C03644=1019.173,313.342,359.557,170.379,50.215,159.769
C03645=1019.180,313.589,359.524,170.385,50.211,159.769
C03646=1019.186,313.837,359.491,170.391,50.208,159.770
C03647=1019.193,314.084,359.457,170.397,50.204,159.770
C03648=1019.200,314.331,359.424,170.404,50.201,159.770
C03649=1019.206,314.579,359.390,170.409,50.197,159.770
C03650=1019.212,314.826,359.357,170.415,50.194,159.770
C03651=1019.219,315.075,359.323,170.421,50.191,159.771
C03652=1019.226,315.322,359.290,170.427,50.187,159.771
C03653=1019.232,315.570,359.256,170.433,50.185,159.771
C03654=1019.239,315.817,359.223,170.439,50.181,159.771
C03655=1019.246,316.065,359.189,170.444,50.178,159.772
C03656=1019.252,316.312,359.156,170.451,50.175,159.772
C03657=1019.259,316.560,359.122,170.457,50.171,159.772
C03658=1019.265,316.807,359.088,170.463,50.168,159.772
C03659=1019.272,317.056,359.055,170.469,50.165,159.773
C03660=1019.279,317.303,359.021,170.475,50.162,159.773
C03661=1019.285,317.551,358.987,170.481,50.158,159.773
C03662=1019.292,317.798,358.954,170.487,50.156,159.773
C03663=1019.299,318.046,358.921,170.493,50.152,159.774
C03664=1019.306,318.294,358.887,170.500,50.149,159.774
C03665=1019.312,318.542,358.853,170.505,50.146,159.774
C03666=1019.319,318.789,358.819,170.512,50.143,159.775
C03667=1019.326,319.036,358.785,170.518,50.139,159.775
C03668=1019.333,319.284,358.752,170.523,50.136,159.775
C03669=1019.339,319.531,358.717,170.530,50.133,159.775
C03670=1019.346,319.779,358.684,170.535,50.130,159.776
C03671=1019.353,320.027,358.651,170.542,50.127,159.776
C03672=1019.360,320.274,358.617,170.549,50.124,159.776
C03673=1019.366,320.522,358.583,170.554,50.121,159.776
C03674=1019.374,320.770,358.549,170.561,50.118,159.777
C03675=1019.381,321.017,358.515,170.566,50.115,159.777
C03676=1019.387,321.264,358.482,170.572,50.111,159.777
C03677=1019.394,321.512,358.447,170.579,50.108,159.778
C03678=1019.401,321.760,358.413,170.585,50.106,159.778
C03679=1019.408,322.009,358.379,170.591,50.103,159.778
C03680=1019.415,322.258,358.344,170.598,50.099,159.779
C03681=1019.422,322.507,358.311,170.603,50.096,159.779
C03682=1019.429,322.756,358.276,170.610,50.093,159.779
C03683=1019.437,323.004,358.242,170.617,50.090,159.780
C03684=1019.443,323.252,358.208,170.622,50.088,159.780
C03685=1019.450,323.498,358.174,170.629,50.084,159.780
C03686=1019.457,323.746,358.141,170.635,50.081,159.781
C03687=1019.463,323.994,358.106,170.642,50.078,159.781
C03688=1019.471,324.241,358.072,170.647,50.075,159.781
C03689=1019.478,324.489,358.038,170.654,50.072,159.782
C03690=1019.485,324.737,358.004,170.661,50.069,159.782
C03691=1019.492,324.985,357.970,170.666,50.066,159.782
C03692=1019.499,325.232,357.935,170.673,50.063,159.783
C03693=1019.506,325.479,357.901,170.680,50.060,159.783
C03694=1019.514,325.727,357.867,170.685,50.058,159.783
C03695=1019.520,325.974,357.832,170.692,50.055,159.784
C03696=1019.528,326.222,357.798,170.699,50.052,159.784
C03697=1019.535,326.469,357.764,170.704,50.049,159.784
C03698=1019.542,326.717,357.730,170.711,50.046,159.785
C03699=1019.548,326.964,357.694,170.718,50.043,159.785
C03700=1019.555,327.212,357.661,170.724,50.041,159.786
C03701=1019.562,327.459,357.625,170.730,50.038,159.786
C03702=1019.569,327.707,357.590,170.737,50.035,159.787
C03703=1019.576,327.954,357.556,170.743,50.032,159.787
C03704=1019.583,328.202,357.521,170.750,50.030,159.787
C03705=1019.590,328.449,357.486,170.756,50.027,159.788
C03706=1019.597,328.697,357.451,170.762,50.024,159.788
C03707=1019.604,328.944,357.417,170.769,50.022,159.789
C03708=1019.610,329.192,357.382,170.776,50.019,159.789
C03709=1019.617,329.439,357.347,170.781,50.016,159.789
C03710=1019.625,329.686,357.312,170.788,50.014,159.790
C03711=1019.632,329.933,357.277,170.795,50.011,159.790
C03712=1019.639,330.182,357.242,170.801,50.009,159.791
C03713=1019.645,330.429,357.207,170.808,50.006,159.791
C03714=1019.653,330.676,357.173,170.814,50.003,159.792
C03715=1019.660,330.924,357.138,170.821,50.000,159.792
C03716=1019.666,331.171,357.103,170.827,49.998,159.793
C03717=1019.673,331.419,357.067,170.834,49.995,159.793
C03718=1019.681,331.666,357.033,170.841,49.992,159.793
C03719=1019.688,331.914,356.997,170.847,49.990,159.794
C03720=1019.695,332.161,356.962,170.853,49.987,159.794
C03721=1019.702,332.408,356.928,170.860,49.985,159.795
C03722=1019.710,332.656,356.892,170.867,49.983,159.796
C03723=1019.716,332.904,356.857,170.873,49.980,159.796
C03724=1019.723,333.151,356.822,170.880,49.978,159.796
C03725=1019.730,333.398,356.786,170.887,49.975,159.797
C03726=1019.738,333.646,356.751,170.893,49.972,159.797
C03727=1019.744,333.893,356.715,170.900,49.970,159.798
C03728=1019.751,334.140,356.680,170.907,49.968,159.798
C03729=1019.758,334.387,356.644,170.914,49.965,159.799
C03730=1019.766,334.635,356.609,170.919,49.963,159.799
C03731=1019.772,334.883,356.574,170.926,49.960,159.800
C03732=1019.779,335.129,356.538,170.933,49.958,159.801
C03733=1019.787,335.377,356.502,170.939,49.956,159.801
C03734=1019.794,335.625,356.467,170.946,49.954,159.802
C03735=1019.801,335.872,356.431,170.953,49.951,159.802
C03736=1019.808,336.120,356.396,170.960,49.948,159.803
C03737=1019.815,336.366,356.360,170.966,49.946,159.803
C03738=1019.823,336.614,356.325,170.973,49.944,159.804
C03739=1019.830,336.860,356.290,170.980,49.941,159.804
C03740=1019.837,337.106,356.253,170.987,49.939,159.805
C03741=1019.844,337.352,356.218,170.993,49.937,159.805
C03742=1019.851,337.599,356.182,171.000,49.935,159.806
C03743=1019.859,337.844,356.148,171.007,49.932,159.806
C03744=1019.866,338.091,356.112,171.014,49.930,159.807
C03745=1019.873,338.336,356.076,171.020,49.928,159.808
C03746=1019.880,338.583,356.040,171.027,49.926,159.808
C03747=1019.887,338.830,356.004,171.034,49.923,159.809
C03748=1019.895,339.078,355.969,171.042,49.921,159.810
C03749=1019.902,339.324,355.933,171.049,49.919,159.810
C03750=1019.909,339.572,355.897,171.055,49.917,159.811
C03751=1019.917,339.819,355.861,171.062,49.915,159.811
C03752=1019.924,340.066,355.824,171.069,49.912,159.812
C03753=1019.931,340.315,355.789,171.076,49.911,159.813
C03754=1019.938,340.561,355.753,171.083,49.908,159.813
C03755=1019.946,340.809,355.717,171.089,49.906,159.814
C03756=1019.952,341.056,355.680,171.096,49.904,159.814
C03757=1019.960,341.303,355.644,171.104,49.902,159.815
C03758=1019.967,341.551,355.608,171.111,49.900,159.816
C03759=1019.974,341.797,355.572,171.118,49.897,159.816
C03760=1019.981,342.045,355.535,171.124,49.896,159.817
C03761=1019.989,342.293,355.499,171.131,49.894,159.817
C03762=1019.996,342.539,355.463,171.139,49.892,159.818
C03763=1020.004,342.786,355.426,171.146,49.889,159.819
C03764=1020.011,343.034,355.389,171.153,49.888,159.820
C03765=1020.018,343.281,355.353,171.160,49.885,159.820
C03766=1020.026,343.528,355.317,171.166,49.884,159.821
C03767=1020.033,343.776,355.280,171.173,49.882,159.821
C03768=1020.040,344.023,355.244,171.181,49.880,159.822
C03769=1020.048,344.269,355.208,171.188,49.877,159.823
C03770=1020.055,344.517,355.171,171.195,49.876,159.824
C03771=1020.062,344.765,355.135,171.202,49.873,159.824
C03772=1020.070,345.011,355.098,171.210,49.872,159.825
C03773=1020.077,345.259,355.061,171.217,49.870,159.826
C03774=1020.085,345.507,355.025,171.223,49.868,159.826
C03775=1020.092,345.753,354.988,171.230,49.866,159.827
C03776=1020.099,346.001,354.951,171.238,49.864,159.828
C03777=1020.107,346.247,354.914,171.245,49.862,159.828
C03778=1020.115,346.495,354.878,171.252,49.860,159.829
C03779=1020.122,346.742,354.841,171.260,49.859,159.830
C03780=1020.130,346.989,354.804,171.267,49.857,159.831
C03781=1020.138,347.236,354.767,171.274,49.854,159.831
C03782=1020.145,347.484,354.731,171.281,49.853,159.832
C03783=1020.152,347.731,354.693,171.289,49.851,159.833
C03784=1020.160,347.978,354.656,171.296,49.849,159.834
C03785=1020.167,348.226,354.619,171.304,49.848,159.834
C03786=1020.175,348.473,354.582,171.310,49.846,159.835
C03787=1020.182,348.720,354.545,171.317,49.844,159.836
C03788=1020.190,348.966,354.508,171.325,49.843,159.837
C03789=1020.197,349.214,354.471,171.332,49.841,159.837
C03790=1020.205,349.461,354.434,171.340,49.839,159.838
C03791=1020.212,349.708,354.397,171.347,49.837,159.839
C03792=1020.220,349.955,354.359,171.354,49.836,159.840
C03793=1020.228,350.202,354.322,171.362,49.834,159.841
C03794=1020.235,350.449,354.285,171.369,49.832,159.841
C03795=1020.242,350.696,354.247,171.376,49.830,159.842
C03796=1020.250,350.943,354.210,171.384,49.829,159.843
C03797=1020.257,351.190,354.173,171.392,49.828,159.844
C03798=1020.265,351.437,354.136,171.399,49.826,159.845
C03799=1020.272,351.682,354.099,171.406,49.824,159.845
C03800=1020.280,351.927,354.062,171.414,49.822,159.846
C03801=1020.288,352.171,354.025,171.421,49.821,159.847
C03802=1020.295,352.416,353.988,171.429,49.820,159.848
C03803=1020.302,352.661,353.951,171.436,49.818,159.849
C03804=1020.310,352.905,353.914,171.444,49.816,159.850
C03805=1020.318,353.150,353.876,171.451,49.814,159.850
C03806=1020.326,353.394,353.839,171.459,49.813,159.851
C03807=1020.334,353.641,353.802,171.466,49.811,159.852
C03808=1020.341,353.888,353.764,171.474,49.810,159.853
C03809=1020.350,354.135,353.726,171.481,49.809,159.854
C03810=1020.357,354.382,353.689,171.489,49.807,159.855
C03811=1020.364,354.629,353.651,171.497,49.806,159.856
C03812=1020.372,354.876,353.613,171.504,49.804,159.856
C03813=1020.380,355.124,353.575,171.512,49.803,159.857
C03814=1020.388,355.370,353.537,171.519,49.801,159.858
C03815=1020.395,355.617,353.500,171.527,49.800,159.859
C03816=1020.403,355.864,353.461,171.535,49.799,159.860
C03817=1020.410,356.111,353.424,171.542,49.797,159.861
C03818=1020.418,356.358,353.386,171.550,49.796,159.862
C03819=1020.427,356.605,353.348,171.557,49.794,159.863
C03820=1020.434,356.852,353.310,171.566,49.793,159.864
C03821=1020.442,357.099,353.271,171.574,49.792,159.865
C03822=1020.450,357.346,353.234,171.582,49.791,159.866
C03823=1020.458,357.594,353.195,171.589,49.789,159.866
C03824=1020.465,357.840,353.157,171.597,49.788,159.867
C03825=1020.474,358.087,353.119,171.604,49.787,159.868
C03826=1020.481,358.334,353.081,171.612,49.785,159.869
C03827=1020.490,358.581,353.043,171.620,49.784,159.870
C03828=1020.497,358.828,353.005,171.628,49.782,159.871
C03829=1020.505,359.075,352.966,171.636,49.781,159.872
C03830=1020.513,359.322,352.928,171.644,49.780,159.873
C03831=1020.521,359.569,352.889,171.652,49.779,159.874
C03832=1020.529,359.815,352.851,171.659,49.778,159.875
C03833=1020.537,360.063,352.812,171.667,49.777,159.876
C03834=1020.544,360.309,352.774,171.676,49.775,159.877
C03835=1020.552,360.556,352.735,171.684,49.774,159.878
C03836=1020.561,360.803,352.697,171.691,49.773,159.879
C03837=1020.568,361.050,352.659,171.699,49.772,159.880
C03838=1020.575,361.298,352.619,171.707,49.771,159.881
C03839=1020.583,361.543,352.580,171.716,49.770,159.882
C03840=1020.591,361.791,352.542,171.724,49.769,159.883
C03841=1020.600,362.038,352.503,171.732,49.768,159.884
C03842=1020.607,362.284,352.465,171.739,49.766,159.885
C03843=1020.616,362.531,352.426,171.747,49.765,159.886
C03844=1020.624,362.778,352.387,171.756,49.764,159.888
C03845=1020.631,363.025,352.349,171.764,49.763,159.889
C03846=1020.639,363.272,352.309,171.772,49.762,159.890
C03847=1020.647,363.519,352.270,171.780,49.762,159.891
C03848=1020.656,363.765,352.231,171.789,49.760,159.892
C03849=1020.664,364.013,352.192,171.796,49.759,159.893
C03850=1020.672,364.258,352.153,171.805,49.759,159.894
C03851=1020.680,364.506,352.115,171.813,49.757,159.895
C03852=1020.688,364.752,352.075,171.821,49.757,159.896
C03853=1020.696,365.000,352.036,171.829,49.755,159.897
C03854=1020.704,365.246,351.997,171.837,49.754,159.898
C03855=1020.713,365.493,351.958,171.846,49.753,159.899
C03856=1020.721,365.740,351.919,171.854,49.752,159.900
C03857=1020.729,365.986,351.880,171.862,49.752,159.902
C03858=1020.737,366.233,351.841,171.871,49.751,159.903
C03859=1020.745,366.482,351.801,171.879,49.750,159.904
C03860=1020.753,366.732,351.762,171.888,49.749,159.905
C03861=1020.762,366.981,351.722,171.896,49.748,159.906
C03862=1020.770,367.231,351.682,171.905,49.747,159.907
C03863=1020.779,367.478,351.643,171.913,49.746,159.908
C03864=1020.787,367.725,351.603,171.921,49.746,159.910
C03865=1020.796,367.971,351.564,171.930,49.744,159.911
C03866=1020.804,368.218,351.524,171.938,49.744,159.912
C03867=1020.812,368.465,351.485,171.947,49.743,159.913
C03868=1020.820,368.712,351.445,171.955,49.742,159.914
C03869=1020.828,368.958,351.406,171.963,49.742,159.916
C03870=1020.836,369.205,351.366,171.973,49.741,159.917
C03871=1020.845,369.451,351.326,171.981,49.741,159.918
C03872=1020.852,369.698,351.286,171.990,49.740,159.919
C03873=1020.861,369.945,351.246,171.998,49.739,159.920
C03874=1020.869,370.192,351.207,172.007,49.738,159.922
C03875=1020.877,370.437,351.167,172.015,49.738,159.923
C03876=1020.885,370.684,351.127,172.023,49.737,159.924
C03877=1020.894,370.932,351.087,172.033,49.736,159.925
C03878=1020.902,371.178,351.046,172.041,49.736,159.927
C03879=1020.911,371.425,351.007,172.050,49.735,159.928
C03880=1020.919,371.671,350.966,172.058,49.734,159.929
C03881=1020.927,371.917,350.927,172.067,49.734,159.930
C03882=1020.936,372.165,350.887,172.076,49.734,159.932
C03883=1020.944,372.411,350.847,172.085,49.733,159.933
C03884=1020.953,372.657,350.807,172.093,49.732,159.934
C03885=1020.961,372.905,350.766,172.102,49.732,159.936
C03886=1020.970,373.151,350.726,172.111,49.731,159.937
C03887=1020.978,373.397,350.686,172.120,49.731,159.938
C03888=1020.987,373.644,350.646,172.129,49.730,159.939
C03889=1020.995,373.890,350.605,172.137,49.730,159.941
C03890=1021.004,374.137,350.566,172.146,49.729,159.942
C03891=1021.012,374.384,350.525,172.155,49.729,159.943
C03892=1021.021,374.630,350.485,172.164,49.728,159.945
C03893=1021.030,374.877,350.444,172.173,49.728,159.946
C03894=1021.038,375.123,350.404,172.182,49.727,159.947
C03895=1021.047,375.371,350.364,172.191,49.727,159.949
C03896=1021.055,375.617,350.324,172.200,49.726,159.950
C03897=1021.064,375.864,350.283,172.209,49.726,159.951
C03898=1021.073,376.110,350.243,172.218,49.725,159.953
C03899=1021.081,376.357,350.202,172.227,49.725,159.954
C03900=1021.089,376.603,350.161,172.236,49.725,159.955
C03901=1021.098,376.850,350.120,172.245,49.725,159.957
C03902=1021.107,377.095,350.079,172.254,49.724,159.958
C03903=1021.116,377.342,350.038,172.263,49.724,159.960
C03904=1021.124,377.588,349.998,172.272,49.724,159.961
C03905=1021.132,377.835,349.957,172.282,49.723,159.962
C03906=1021.141,378.081,349.915,172.290,49.723,159.964
C03907=1021.150,378.328,349.875,172.300,49.723,159.965
C03908=1021.159,378.575,349.834,172.309,49.723,159.967
C03909=1021.167,378.820,349.792,172.319,49.723,159.968
C03910=1021.176,379.067,349.751,172.327,49.723,159.970
C03911=1021.185,379.314,349.710,172.337,49.722,159.971
C03912=1021.193,379.560,349.669,172.346,49.722,159.973
C03913=1021.202,379.806,349.628,172.356,49.722,159.974
C03914=1021.211,380.053,349.587,172.364,49.722,159.975
C03915=1021.219,380.299,349.546,172.374,49.722,159.977
C03916=1021.228,380.545,349.504,172.383,49.721,159.978
C03917=1021.237,380.792,349.463,172.393,49.721,159.980
C03918=1021.246,381.038,349.421,172.403,49.721,159.982
C03919=1021.256,381.310,349.376,172.412,49.721,159.983
C03920=1021.265,381.581,349.331,172.423,49.721,159.985
C03921=1021.276,381.852,349.285,172.434,49.721,159.986
C03922=1021.285,382.124,349.239,172.444,49.721,159.988
C03923=1021.294,382.370,349.197,172.453,49.721,159.990
C03924=1021.303,382.617,349.156,172.463,49.721,159.991
C03925=1021.313,382.863,349.115,172.473,49.721,159.993
C03926=1021.322,383.109,349.073,172.482,49.721,159.994
C03927=1021.331,383.356,349.031,172.492,49.720,159.996
C03928=1021.339,383.602,348.990,172.502,49.721,159.997
C03929=1021.348,383.848,348.948,172.511,49.720,159.999
C03930=1021.357,384.095,348.906,172.521,49.721,160.001
C03931=1021.367,384.341,348.865,172.531,49.721,160.002
C03932=1021.376,384.587,348.823,172.540,49.721,160.004
C03933=1021.385,384.833,348.782,172.550,49.721,160.005
C03934=1021.394,385.080,348.740,172.560,49.721,160.007
C03935=1021.403,385.326,348.698,172.570,49.721,160.008
C03936=1021.412,385.573,348.656,172.580,49.721,160.010
C03937=1021.421,385.819,348.614,172.589,49.721,160.012
C03938=1021.430,386.065,348.572,172.599,49.721,160.013
C03939=1021.440,386.311,348.529,172.609,49.721,160.015
C03940=1021.449,386.558,348.488,172.619,49.722,160.017
C03941=1021.458,386.803,348.445,172.629,49.722,160.018
C03942=1021.467,387.050,348.403,172.638,49.722,160.020
C03943=1021.477,387.296,348.361,172.648,49.723,160.022
C03944=1021.486,387.542,348.319,172.658,49.723,160.023
C03945=1021.495,387.788,348.277,172.669,49.723,160.025
C03946=1021.505,388.035,348.234,172.679,49.723,160.027
C03947=1021.513,388.281,348.192,172.689,49.723,160.028
C03948=1021.522,388.527,348.149,172.699,49.724,160.030
C03949=1021.531,388.773,348.107,172.709,49.724,160.032
C03950=1021.541,389.019,348.064,172.719,49.725,160.034
C03951=1021.550,389.265,348.021,172.729,49.725,160.035
C03952=1021.559,389.512,347.978,172.740,49.725,160.037
C03953=1021.569,389.757,347.936,172.749,49.725,160.039
C03954=1021.578,390.003,347.893,172.760,49.726,160.041
C03955=1021.588,390.250,347.850,172.770,49.726,160.042
C03956=1021.596,390.496,347.807,172.781,49.727,160.044
C03957=1021.606,390.742,347.765,172.791,49.727,160.046
C03958=1021.615,390.988,347.722,172.801,49.727,160.048
C03959=1021.625,391.234,347.679,172.811,49.728,160.050
C03960=1021.634,391.480,347.637,172.822,49.728,160.051
C03961=1021.644,391.727,347.593,172.832,49.729,160.053
C03962=1021.653,391.972,347.550,172.842,49.730,160.055
C03963=1021.663,392.218,347.508,172.853,49.730,160.057
C03964=1021.671,392.464,347.464,172.863,49.731,160.059
C03965=1021.682,392.710,347.421,172.873,49.731,160.060
C03966=1021.691,392.957,347.378,172.884,49.732,160.062
C03967=1021.700,393.202,347.334,172.895,49.732,160.064
C03968=1021.710,393.449,347.292,172.905,49.733,160.066
C03969=1021.720,393.694,347.248,172.916,49.734,160.068
C03970=1021.729,393.940,347.205,172.926,49.734,160.070
C03971=1021.739,394.186,347.162,172.937,49.734,160.072
C03972=1021.748,394.432,347.117,172.948,49.735,160.074
C03973=1021.758,394.679,347.075,172.958,49.736,160.076
C03974=1021.767,394.924,347.031,172.969,49.737,160.078
C03975=1021.777,395.170,346.987,172.979,49.737,160.079
C03976=1021.787,395.416,346.944,172.990,49.738,160.081
C03977=1021.796,395.663,346.901,173.001,49.739,160.083
C03978=1021.806,395.909,346.857,173.012,49.739,160.085
C03979=1021.819,396.217,346.802,173.026,49.740,160.088
C03980=1021.831,396.525,346.747,173.039,49.742,160.090
C03981=1021.843,396.834,346.693,173.053,49.743,160.093
C03982=1021.855,397.142,346.637,173.067,49.744,160.095
C03983=1021.865,397.388,346.593,173.078,49.744,160.097
C03984=1021.875,397.634,346.550,173.088,49.745,160.099
C03985=1021.884,397.880,346.506,173.100,49.746,160.101
C03986=1021.895,398.126,346.461,173.110,49.747,160.103
C03987=1021.904,398.372,346.417,173.122,49.748,160.105
C03988=1021.914,398.618,346.373,173.133,49.748,160.107
C03989=1021.924,398.863,346.329,173.144,49.750,160.110
C03990=1021.934,399.109,346.285,173.155,49.750,160.111
C03991=1021.944,399.355,346.241,173.167,49.751,160.114
C03992=1021.954,399.601,346.196,173.177,49.752,160.116
C03993=1021.964,399.847,346.151,173.189,49.753,160.118
C03994=1021.974,400.093,346.108,173.200,49.754,160.120
C03995=1021.984,400.338,346.063,173.212,49.755,160.122
C03996=1021.993,400.584,346.019,173.222,49.756,160.124
C03997=1022.004,400.830,345.974,173.234,49.757,160.126
C03998=1022.014,401.076,345.929,173.245,49.758,160.128
C03999=1022.024,401.321,345.885,173.257,49.759,160.131
C04000=1022.033,401.567,345.840,173.269,49.760,160.133
C04001=1022.043,401.814,345.795,173.279,49.762,160.135
C04002=1022.053,402.059,345.751,173.291,49.763,160.137
C04003=1022.063,402.304,345.706,173.302,49.764,160.139
C04004=1022.074,402.550,345.661,173.314,49.765,160.141
C04005=1022.084,402.795,345.616,173.326,49.766,160.144
C04006=1022.093,403.041,345.571,173.338,49.767,160.146
C04007=1022.104,403.287,345.526,173.349,49.768,160.148
C04008=1022.114,403.532,345.481,173.361,49.769,160.150
C04009=1022.125,403.778,345.436,173.373,49.770,160.152
C04010=1022.134,404.024,345.391,173.385,49.772,160.155
C04011=1022.145,404.270,345.345,173.396,49.773,160.157
C04012=1022.155,404.515,345.301,173.408,49.774,160.159
C04013=1022.165,404.761,345.255,173.420,49.776,160.162
C04014=1022.176,405.006,345.210,173.431,49.777,160.164
C04015=1022.186,405.252,345.165,173.443,49.778,160.166
C04016=1022.196,405.497,345.120,173.455,49.779,160.168
C04017=1022.206,405.743,345.075,173.467,49.781,160.171
C04018=1022.217,405.989,345.029,173.479,49.782,160.173
C04019=1022.227,406.235,344.983,173.491,49.783,160.175
C04020=1022.237,406.480,344.938,173.503,49.785,160.178
C04021=1022.249,406.725,344.893,173.516,49.786,160.180
C04022=1022.259,406.971,344.847,173.527,49.787,160.182
C04023=1022.270,407.217,344.801,173.539,49.789,160.185
C04024=1022.280,407.462,344.756,173.551,49.790,160.187
C04025=1022.290,407.708,344.710,173.563,49.792,160.190
C04026=1022.301,407.954,344.665,173.576,49.793,160.192
C04027=1022.312,408.199,344.620,173.588,49.795,160.194
C04028=1022.323,408.445,344.574,173.600,49.796,160.197
C04029=1022.333,408.690,344.528,173.613,49.798,160.199
C04030=1022.344,408.936,344.482,173.625,49.799,160.202
C04031=1022.354,409.181,344.436,173.637,49.801,160.204
C04032=1022.365,409.427,344.390,173.650,49.802,160.207
C04033=1022.376,409.672,344.343,173.662,49.803,160.209
C04034=1022.387,409.918,344.297,173.675,49.806,160.212
C04035=1022.397,410.163,344.252,173.688,49.807,160.214
C04036=1022.407,410.408,344.204,173.700,49.808,160.216
C04037=1022.418,410.654,344.158,173.712,49.811,160.219
C04038=1022.429,410.899,344.112,173.725,49.812,160.222
C04039=1022.444,411.231,344.049,173.743,49.814,160.225
C04040=1022.458,411.561,343.987,173.760,49.816,160.228
C04041=1022.473,411.893,343.924,173.776,49.819,160.232
C04042=1022.488,412.224,343.861,173.794,49.821,160.235
C04043=1022.498,412.470,343.814,173.807,49.823,160.238
C04044=1022.509,412.715,343.768,173.819,49.825,160.241
C04045=1022.520,412.960,343.721,173.833,49.826,160.243
C04046=1022.531,413.206,343.674,173.846,49.828,160.246
C04047=1022.542,413.451,343.628,173.858,49.830,160.248
C04048=1022.554,413.697,343.581,173.871,49.831,160.251
C04049=1022.564,413.942,343.533,173.885,49.833,160.254
C04050=1022.575,414.187,343.487,173.897,49.835,160.256
C04051=1022.587,414.433,343.440,173.911,49.837,160.259
C04052=1022.598,414.678,343.393,173.924,49.839,160.262
C04053=1022.609,414.923,343.346,173.937,49.840,160.264
C04054=1022.621,415.169,343.299,173.950,49.842,160.267
C04055=1022.631,415.414,343.252,173.964,49.845,160.270
C04056=1022.643,415.659,343.204,173.977,49.847,160.273
C04057=1022.653,415.905,343.157,173.990,49.848,160.275
C04058=1022.665,416.150,343.109,174.004,49.851,160.278
C04059=1022.676,416.395,343.062,174.017,49.852,160.281
C04060=1022.687,416.640,343.014,174.031,49.855,160.284
C04061=1022.698,416.886,342.967,174.044,49.857,160.286
C04062=1022.709,417.131,342.919,174.057,49.859,160.289
C04063=1022.721,417.375,342.872,174.071,49.861,160.292
C04064=1022.731,417.621,342.824,174.085,49.863,160.295
C04065=1022.743,417.866,342.776,174.098,49.865,160.298
C04066=1022.755,418.111,342.729,174.112,49.867,160.301
C04067=1022.766,418.357,342.680,174.126,49.869,160.304
C04068=1022.778,418.602,342.633,174.140,49.871,160.306
C04069=1022.788,418.847,342.585,174.154,49.873,160.309
C04070=1022.800,419.092,342.537,174.168,49.875,160.312
C04071=1022.811,419.337,342.489,174.182,49.878,160.315
C04072=1022.823,419.582,342.441,174.195,49.880,160.318
C04073=1022.835,419.827,342.393,174.209,49.882,160.321
C04074=1022.846,420.072,342.345,174.224,49.884,160.324
C04075=1022.858,420.317,342.297,174.238,49.886,160.327
C04076=1022.870,420.563,342.248,174.251,49.888,160.330
C04077=1022.882,420.808,342.200,174.265,49.891,160.333
C04078=1022.894,421.053,342.153,174.280,49.893,160.336
C04079=1022.905,421.298,342.104,174.294,49.895,160.339
C04080=1022.917,421.543,342.056,174.308,49.898,160.342
C04081=1022.929,421.789,342.007,174.323,49.900,160.345
C04082=1022.940,422.034,341.958,174.337,49.902,160.348
C04083=1022.952,422.278,341.910,174.352,49.905,160.351
C04084=1022.964,422.523,341.861,174.366,49.907,160.354
C04085=1022.975,422.769,341.812,174.380,49.910,160.357
C04086=1022.987,423.013,341.764,174.395,49.912,160.360
C04087=1022.999,423.258,341.715,174.409,49.915,160.364
C04088=1023.011,423.503,341.665,174.424,49.917,160.367
C04089=1023.023,423.748,341.617,174.439,49.919,160.370
C04090=1023.034,423.993,341.568,174.453,49.922,160.373
C04091=1023.047,424.238,341.519,174.469,49.924,160.376
C04092=1023.059,424.483,341.470,174.483,49.927,160.379
C04093=1023.071,424.728,341.421,174.498,49.929,160.382
C04094=1023.083,424.972,341.372,174.513,49.932,160.386
C04095=1023.095,425.217,341.322,174.528,49.935,160.389
C04096=1023.107,425.463,341.273,174.543,49.937,160.392
C04097=1023.120,425.708,341.224,174.558,49.940,160.395
C04098=1023.131,425.952,341.174,174.573,49.942,160.399
C04099=1023.145,426.222,341.120,174.590,49.945,160.402
C04100=1023.158,426.491,341.065,174.607,49.948,160.406
C04101=1023.171,426.761,341.010,174.623,49.951,160.410
C04102=1023.185,427.031,340.956,174.640,49.954,160.413
C04103=1023.197,427.275,340.906,174.655,49.957,160.417
C04104=1023.209,427.520,340.856,174.670,49.960,160.420
C04105=1023.221,427.764,340.806,174.686,49.963,160.423
C04106=1023.234,428.009,340.756,174.701,49.965,160.427
C04107=1023.246,428.254,340.706,174.717,49.968,160.430
C04108=1023.258,428.499,340.656,174.732,49.971,160.434
C04109=1023.271,428.744,340.605,174.749,49.974,160.437
C04110=1023.284,428.988,340.556,174.764,49.977,160.441
C04111=1023.296,429.233,340.506,174.780,49.979,160.444
C04112=1023.308,429.478,340.456,174.796,49.982,160.447
C04113=1023.321,429.722,340.405,174.811,49.985,160.451
C04114=1023.333,429.967,340.355,174.827,49.988,160.454
C04115=1023.346,430.212,340.305,174.843,49.990,160.458
C04116=1023.358,430.456,340.254,174.859,49.994,160.461
C04117=1023.371,430.700,340.204,174.875,49.997,160.465
C04118=1023.384,430.945,340.154,174.892,50.000,160.469
C04119=1023.397,431.190,340.103,174.907,50.003,160.472
C04120=1023.409,431.434,340.052,174.924,50.006,160.476
C04121=1023.422,431.678,340.002,174.940,50.008,160.479
C04122=1023.434,431.923,339.951,174.956,50.012,160.483
C04123=1023.448,432.168,339.901,174.973,50.015,160.487
C04124=1023.461,432.413,339.850,174.989,50.017,160.490
C04125=1023.474,432.657,339.799,175.005,50.021,160.494
C04126=1023.487,432.901,339.748,175.022,50.024,160.497
C04127=1023.500,433.146,339.697,175.038,50.027,160.501
C04128=1023.513,433.390,339.646,175.055,50.030,160.505
C04129=1023.525,433.636,339.594,175.072,50.033,160.509
C04130=1023.538,433.879,339.543,175.088,50.036,160.512
C04131=1023.551,434.124,339.492,175.105,50.040,160.516
C04132=1023.564,434.369,339.440,175.122,50.043,160.520
C04133=1023.577,434.612,339.389,175.139,50.046,160.524
C04134=1023.591,434.857,339.338,175.156,50.049,160.528
C04135=1023.603,435.101,339.286,175.172,50.053,160.531
C04136=1023.617,435.345,339.234,175.190,50.056,160.535
C04137=1023.630,435.590,339.183,175.206,50.059,160.539
C04138=1023.644,435.834,339.131,175.224,50.062,160.543
C04139=1023.660,436.152,339.064,175.247,50.067,160.548
C04140=1023.678,436.468,338.997,175.269,50.071,160.553
C04141=1023.695,436.786,338.929,175.291,50.076,160.558
C04142=1023.713,437.103,338.862,175.314,50.080,160.563
C04143=1023.726,437.347,338.810,175.332,50.083,160.567
C04144=1023.740,437.592,338.758,175.349,50.087,160.571
C04145=1023.753,437.836,338.706,175.366,50.090,160.575
C04146=1023.766,438.080,338.653,175.384,50.093,160.579
C04147=1023.780,438.324,338.601,175.402,50.097,160.584
C04148=1023.794,438.568,338.548,175.420,50.101,160.587
C04149=1023.807,438.812,338.496,175.438,50.104,160.592
C04150=1023.820,439.056,338.443,175.456,50.108,160.596
C04151=1023.834,439.301,338.391,175.474,50.111,160.600
C04152=1023.848,439.545,338.338,175.492,50.115,160.604
C04153=1023.862,439.788,338.286,175.510,50.118,160.608
C04154=1023.875,440.032,338.232,175.528,50.122,160.612
C04155=1023.889,440.277,338.180,175.547,50.126,160.617
C04156=1023.903,440.521,338.128,175.565,50.130,160.621
C04157=1023.918,440.765,338.075,175.583,50.133,160.625
C04158=1023.931,441.009,338.022,175.602,50.137,160.629
C04159=1023.946,441.268,337.966,175.621,50.141,160.634
C04160=1023.961,441.529,337.909,175.641,50.144,160.638
C04161=1023.976,441.789,337.852,175.661,50.148,160.643
C04162=1023.991,442.047,337.795,175.680,50.152,160.647
C04163=1023.596,440.124,337.880,175.526,50.187,160.632
C04164=1023.583,439.880,337.933,175.508,50.184,160.628
C04165=1023.569,439.636,337.986,175.490,50.180,160.624
C04166=1023.555,439.391,338.038,175.472,50.177,160.620
C04167=1023.541,439.147,338.091,175.453,50.174,160.615
C04168=1023.528,438.903,338.144,175.436,50.170,160.611
C04169=1023.514,438.659,338.196,175.417,50.167,160.607
C04170=1023.501,438.415,338.248,175.400,50.163,160.603
C04171=1023.487,438.171,338.300,175.382,50.160,160.599
C04172=1023.474,437.927,338.353,175.364,50.157,160.595
C04173=1023.460,437.682,338.406,175.347,50.154,160.591
C04174=1023.446,437.438,338.458,175.329,50.150,160.587
C04175=1023.433,437.194,338.509,175.311,50.147,160.583
C04176=1023.419,436.949,338.561,175.294,50.144,160.579
C04177=1023.406,436.705,338.613,175.276,50.140,160.575
C04178=1023.393,436.461,338.665,175.259,50.137,160.571
C04179=1023.379,436.217,338.717,175.242,50.133,160.567
C04180=1023.366,435.973,338.769,175.225,50.130,160.564
C04181=1023.353,435.728,338.820,175.207,50.127,160.560
C04182=1023.340,435.483,338.872,175.190,50.124,160.556
C04183=1023.327,435.240,338.924,175.173,50.121,160.552
C04184=1023.314,434.995,338.975,175.156,50.118,160.548
C04185=1023.300,434.751,339.027,175.139,50.115,160.544
C04186=1023.287,434.506,339.078,175.122,50.111,160.540
C04187=1023.274,434.262,339.129,175.105,50.108,160.537
C04188=1023.261,434.017,339.181,175.088,50.105,160.533
C04189=1023.248,433.773,339.231,175.071,50.102,160.529
C04190=1023.235,433.529,339.283,175.055,50.099,160.525
C04191=1023.222,433.285,339.334,175.038,50.096,160.522
C04192=1023.209,433.040,339.385,175.021,50.093,160.518
C04193=1023.197,432.795,339.437,175.005,50.090,160.514
C04194=1023.184,432.551,339.488,174.988,50.087,160.511
C04195=1023.170,432.306,339.538,174.972,50.084,160.507
C04196=1023.158,432.062,339.589,174.956,50.081,160.503
C04197=1023.144,431.817,339.640,174.939,50.078,160.500
C04198=1023.132,431.572,339.690,174.923,50.075,160.496
C04199=1023.119,431.328,339.741,174.906,50.072,160.492
C04200=1023.106,431.083,339.792,174.891,50.069,160.489
C04201=1023.093,430.839,339.842,174.874,50.067,160.485
C04202=1023.081,430.595,339.893,174.858,50.064,160.482
C04203=1023.068,430.350,339.943,174.841,50.061,160.478
C04204=1023.054,430.093,339.995,174.825,50.058,160.475
C04205=1023.042,429.838,340.048,174.809,50.055,160.471
C04206=1023.028,429.583,340.101,174.792,50.052,160.467
C04207=1023.015,429.327,340.153,174.775,50.050,160.464
C04208=1023.003,429.082,340.203,174.760,50.047,160.460
C04209=1022.991,428.837,340.253,174.744,50.044,160.457
C04210=1022.978,428.592,340.303,174.728,50.041,160.453
C04211=1022.966,428.348,340.353,174.712,50.039,160.450
C04212=1022.954,428.103,340.404,174.697,50.036,160.447
C04213=1022.941,427.858,340.454,174.681,50.033,160.443
C04214=1022.928,427.613,340.503,174.666,50.031,160.440
C04215=1022.916,427.369,340.553,174.650,50.028,160.436
C04216=1022.900,427.040,340.620,174.630,50.025,160.432
C04217=1022.884,426.711,340.687,174.609,50.020,160.427
C04218=1022.867,426.383,340.753,174.589,50.017,160.423
C04219=1022.852,426.055,340.820,174.568,50.014,160.419
C04220=1022.839,425.810,340.869,174.554,50.011,160.416
C04221=1022.827,425.565,340.919,174.538,50.008,160.412
C04222=1022.816,425.320,340.968,174.523,50.006,160.409
C04223=1022.803,425.075,341.018,174.508,50.004,160.406
C04224=1022.791,424.830,341.066,174.493,50.001,160.402
C04225=1022.779,424.586,341.116,174.479,49.999,160.399
C04226=1022.767,424.340,341.165,174.463,49.996,160.396
C04227=1022.755,424.096,341.213,174.448,49.994,160.393
C04228=1022.743,423.850,341.263,174.434,49.992,160.390
C04229=1022.731,423.606,341.311,174.419,49.989,160.387
C04230=1022.719,423.361,341.360,174.404,49.987,160.383
C04231=1022.707,423.116,341.410,174.390,49.984,160.380
C04232=1022.695,422.871,341.458,174.375,49.982,160.377
C04233=1022.684,422.626,341.507,174.361,49.980,160.374
C04234=1022.672,422.380,341.556,174.346,49.978,160.371
C04235=1022.660,422.136,341.604,174.332,49.975,160.368
C04236=1022.649,421.891,341.653,174.317,49.973,160.365
C04237=1022.637,421.646,341.701,174.303,49.970,160.362
C04238=1022.625,421.401,341.750,174.288,49.969,160.359
C04239=1022.614,421.155,341.798,174.275,49.966,160.356
C04240=1022.602,420.911,341.847,174.260,49.965,160.353
C04241=1022.590,420.666,341.895,174.246,49.962,160.350
C04242=1022.579,420.421,341.943,174.232,49.960,160.347
C04243=1022.567,420.175,341.991,174.217,49.958,160.344
C04244=1022.555,419.931,342.040,174.203,49.955,160.341
C04245=1022.544,419.686,342.087,174.189,49.953,160.338
C04246=1022.532,419.441,342.135,174.176,49.951,160.335
C04247=1022.521,419.195,342.183,174.161,49.950,160.332
C04248=1022.509,418.950,342.231,174.147,49.947,160.329
C04249=1022.498,418.705,342.279,174.134,49.945,160.326
C04250=1022.486,418.460,342.327,174.120,49.943,160.324
C04251=1022.474,418.215,342.375,174.106,49.941,160.321
C04252=1022.463,417.969,342.422,174.093,49.939,160.318
C04253=1022.451,417.724,342.470,174.078,49.937,160.315
C04254=1022.441,417.479,342.518,174.064,49.935,160.312
C04255=1022.429,417.234,342.566,174.051,49.933,160.309
C04256=1022.418,416.988,342.613,174.037,49.932,160.307
C04257=1022.406,416.743,342.661,174.023,49.929,160.304
C04258=1022.395,416.498,342.707,174.010,49.928,160.301
C04259=1022.384,416.253,342.756,173.997,49.926,160.298
C04260=1022.373,416.007,342.803,173.984,49.923,160.295
C04261=1022.362,415.762,342.851,173.970,49.922,160.293
C04262=1022.351,415.517,342.898,173.957,49.920,160.290
C04263=1022.340,415.272,342.945,173.944,49.918,160.287
C04264=1022.329,415.026,342.993,173.930,49.916,160.285
C04265=1022.318,414.781,343.039,173.917,49.915,160.282
C04266=1022.306,414.536,343.086,173.903,49.913,160.279
C04267=1022.295,414.291,343.133,173.890,49.911,160.277
C04268=1022.284,414.045,343.180,173.878,49.909,160.274
C04269=1022.273,413.800,343.226,173.864,49.907,160.271
C04270=1022.262,413.554,343.274,173.851,49.906,160.268
C04271=1022.251,413.309,343.321,173.837,49.904,160.266
C04272=1022.240,413.063,343.368,173.825,49.902,160.263
C04273=1022.229,412.818,343.414,173.812,49.901,160.261
C04274=1022.218,412.573,343.460,173.799,49.899,160.258
C04275=1022.207,412.328,343.507,173.787,49.898,160.256
C04276=1022.192,411.994,343.571,173.769,49.895,160.252
C04277=1022.178,411.661,343.633,173.752,49.893,160.248
C04278=1022.163,411.326,343.697,173.734,49.891,160.245
C04279=1022.149,410.993,343.760,173.717,49.888,160.241
C04280=1022.138,410.748,343.806,173.704,49.887,160.239
C04281=1022.127,410.501,343.853,173.692,49.886,160.237
C04282=1022.116,410.256,343.899,173.678,49.884,160.234
C04283=1022.105,410.011,343.945,173.666,49.882,160.231
C04284=1022.094,409.766,343.992,173.653,49.881,160.229
C04285=1022.084,409.520,344.038,173.641,49.880,160.227
C04286=1022.074,409.274,344.084,173.628,49.878,160.224
C04287=1022.063,409.029,344.130,173.616,49.877,160.222
C04288=1022.053,408.783,344.176,173.604,49.875,160.219
C04289=1022.041,408.538,344.221,173.591,49.874,160.217
C04290=1022.031,408.292,344.267,173.579,49.873,160.214
C04291=1022.020,408.047,344.313,173.567,49.871,160.212
C04292=1022.010,407.802,344.359,173.554,49.870,160.210
C04293=1021.999,407.556,344.405,173.542,49.868,160.207
C04294=1021.989,407.310,344.450,173.531,49.867,160.205
C04295=1021.978,407.065,344.495,173.518,49.866,160.202
C04296=1021.967,406.819,344.541,173.506,49.864,160.200
C04297=1021.957,406.574,344.586,173.494,49.863,160.198
C04298=1021.947,406.328,344.632,173.482,49.862,160.195
C04299=1021.936,406.082,344.678,173.469,49.861,160.193
C04300=1021.926,405.836,344.723,173.457,49.860,160.191
C04301=1021.915,405.592,344.768,173.445,49.858,160.188
C04302=1021.905,405.345,344.813,173.434,49.857,160.186
C04303=1021.894,405.100,344.859,173.422,49.856,160.184
C04304=1021.884,404.854,344.904,173.410,49.854,160.182
C04305=1021.874,404.608,344.949,173.398,49.853,160.179
C04306=1021.863,404.363,344.994,173.386,49.853,160.177
C04307=1021.853,404.117,345.039,173.374,49.851,160.175
C04308=1021.843,403.872,345.084,173.362,49.850,160.173
C04309=1021.833,403.625,345.129,173.350,49.849,160.170
C04310=1021.823,403.381,345.175,173.339,49.848,160.168
C04311=1021.813,403.134,345.220,173.327,49.847,160.166
C04312=1021.802,402.889,345.264,173.315,49.846,160.164
C04313=1021.792,402.644,345.309,173.303,49.845,160.161
C04314=1021.782,402.397,345.354,173.292,49.844,160.159
C04315=1021.772,402.152,345.399,173.281,49.842,160.157
C04316=1021.763,401.906,345.444,173.270,49.842,160.155
C04317=1021.752,401.660,345.489,173.258,49.841,160.153
C04318=1021.742,401.415,345.533,173.247,49.840,160.151
C04319=1021.732,401.170,345.578,173.235,49.839,160.148
C04320=1021.723,400.923,345.622,173.223,49.838,160.146
C04321=1021.712,400.677,345.667,173.212,49.837,160.144
C04322=1021.702,400.432,345.711,173.200,49.836,160.142
C04323=1021.693,400.186,345.755,173.190,49.835,160.140
C04324=1021.683,399.940,345.800,173.178,49.834,160.138
C04325=1021.672,399.695,345.845,173.167,49.833,160.136
C04326=1021.663,399.449,345.889,173.155,49.832,160.134
C04327=1021.653,399.203,345.933,173.144,49.832,160.132
C04328=1021.643,398.957,345.977,173.133,49.830,160.130
C04329=1021.633,398.711,346.021,173.122,49.830,160.128
C04330=1021.623,398.466,346.066,173.111,49.829,160.125
C04331=1021.613,398.219,346.110,173.099,49.828,160.123
C04332=1021.604,397.973,346.154,173.089,49.827,160.121
C04333=1021.594,397.727,346.197,173.077,49.827,160.119
C04334=1021.584,397.482,346.242,173.066,49.826,160.117
C04335=1021.574,397.236,346.286,173.056,49.825,160.115
C04336=1021.562,396.925,346.341,173.042,49.824,160.113
C04337=1021.549,396.614,346.396,173.028,49.823,160.110
C04338=1021.537,396.303,346.452,173.014,49.822,160.108
C04339=1021.525,395.992,346.507,173.000,49.822,160.105
C04340=1021.514,395.746,346.551,172.990,49.821,160.104
C04341=1021.506,395.500,346.594,172.979,49.821,160.102
C04342=1021.496,395.255,346.637,172.967,49.820,160.100
C04343=1021.486,395.009,346.681,172.957,49.819,160.098
C04344=1021.476,394.763,346.725,172.946,49.819,160.096
C04345=1021.466,394.516,346.768,172.936,49.818,160.094
C04346=1021.458,394.271,346.811,172.924,49.818,160.092
C04347=1021.447,394.025,346.855,172.914,49.817,160.090
C04348=1021.438,393.778,346.898,172.903,49.817,160.088
C04349=1021.429,393.533,346.941,172.893,49.816,160.086
C04350=1021.419,393.287,346.984,172.882,49.816,160.084
C04351=1021.410,393.040,347.028,172.871,49.815,160.082
C04352=1021.400,392.795,347.071,172.862,49.814,160.081
C04353=1021.391,392.549,347.115,172.850,49.814,160.079
C04354=1021.382,392.303,347.157,172.840,49.814,160.077
C04355=1021.372,392.056,347.200,172.829,49.813,160.075
C04356=1021.362,391.811,347.244,172.819,49.813,160.073
C04357=1021.353,391.565,347.287,172.809,49.812,160.072
C04358=1021.343,391.318,347.329,172.798,49.812,160.070
C04359=1021.334,391.072,347.372,172.788,49.811,160.068
C04360=1021.324,390.826,347.415,172.778,49.811,160.066
C04361=1021.315,390.580,347.457,172.767,49.811,160.064
C04362=1021.306,390.333,347.500,172.757,49.810,160.063
C04363=1021.296,390.088,347.544,172.747,49.810,160.061
C04364=1021.287,389.842,347.585,172.736,49.810,160.059
C04365=1021.278,389.595,347.628,172.726,49.810,160.057
C04366=1021.269,389.349,347.671,172.716,49.810,160.056
C04367=1021.260,389.104,347.714,172.706,49.809,160.054
C04368=1021.250,388.857,347.756,172.695,49.809,160.052
C04369=1021.241,388.611,347.799,172.685,49.809,160.050
C04370=1021.231,388.366,347.841,172.675,49.808,160.049
C04371=1021.223,388.118,347.884,172.666,49.808,160.047
C04372=1021.213,387.873,347.926,172.656,49.808,160.045
C04373=1021.204,387.627,347.969,172.645,49.808,160.044
C04374=1021.195,387.380,348.011,172.635,49.808,160.042
C04375=1021.185,387.134,348.053,172.625,49.807,160.040
C04376=1021.177,386.888,348.095,172.616,49.808,160.039
C04377=1021.167,386.642,348.137,172.606,49.807,160.037
C04378=1021.158,386.396,348.179,172.596,49.807,160.035
C04379=1021.149,386.150,348.222,172.585,49.807,160.034
C04380=1021.140,385.903,348.264,172.575,49.807,160.032
C04381=1021.130,385.657,348.306,172.566,49.807,160.030
C04382=1021.121,385.411,348.348,172.556,49.807,160.029
C04383=1021.112,385.164,348.390,172.546,49.807,160.027
C04384=1021.104,384.918,348.431,172.536,49.807,160.026
C04385=1021.095,384.672,348.473,172.526,49.807,160.024
C04386=1021.086,384.425,348.515,172.517,49.807,160.022
C04387=1021.077,384.179,348.556,172.507,49.807,160.021
C04388=1021.067,383.933,348.598,172.497,49.807,160.019
C04389=1021.058,383.687,348.640,172.488,49.807,160.018
C04390=1021.049,383.441,348.682,172.478,49.807,160.016
C04391=1021.040,383.194,348.723,172.469,49.807,160.015
C04392=1021.031,382.947,348.764,172.459,49.807,160.013
C04393=1021.022,382.701,348.806,172.449,49.807,160.011
C04394=1021.013,382.455,348.847,172.440,49.808,160.010
C04395=1021.004,382.209,348.889,172.430,49.808,160.009
C04396=1020.994,381.934,348.935,172.419,49.808,160.007
C04397=1020.984,381.661,348.981,172.408,49.808,160.005
C04398=1020.975,381.387,349.027,172.398,49.809,160.003
C04399=1020.964,381.113,349.073,172.387,49.809,160.002
C04400=1020.956,380.867,349.114,172.379,49.809,160.000
C04401=1020.947,380.621,349.156,172.369,49.809,159.999
C04402=1020.938,380.374,349.196,172.360,49.809,159.997
C04403=1020.929,380.128,349.238,172.350,49.810,159.996
C04404=1020.920,379.882,349.279,172.341,49.810,159.994
C04405=1020.912,379.635,349.320,172.331,49.810,159.993
C04406=1020.903,379.389,349.362,172.321,49.811,159.991
C04407=1020.894,379.142,349.403,172.313,49.811,159.990
C04408=1020.885,378.896,349.443,172.303,49.811,159.989
C04409=1020.876,378.649,349.485,172.294,49.811,159.987
C04410=1020.868,378.403,349.525,172.284,49.812,159.986
C04411=1020.859,378.157,349.567,172.275,49.812,159.984
C04412=1020.851,377.910,349.608,172.266,49.812,159.983
C04413=1020.842,377.664,349.648,172.257,49.813,159.981
C04414=1020.833,377.417,349.689,172.248,49.813,159.980
C04415=1020.825,377.171,349.730,172.238,49.813,159.979
C04416=1020.816,376.924,349.771,172.230,49.813,159.977
C04417=1020.808,376.678,349.812,172.221,49.814,159.976
C04418=1020.800,376.431,349.853,172.211,49.814,159.974
C04419=1020.791,376.185,349.893,172.202,49.815,159.973
C04420=1020.782,375.938,349.934,172.193,49.815,159.972
C04421=1020.774,375.692,349.974,172.184,49.816,159.970
C04422=1020.765,375.445,350.015,172.175,49.816,159.969
C04423=1020.756,375.199,350.055,172.167,49.817,159.968
C04424=1020.748,374.952,350.096,172.157,49.817,159.966
C04425=1020.739,374.705,350.135,172.148,49.818,159.965
C04426=1020.731,374.458,350.176,172.139,49.818,159.964
C04427=1020.722,374.212,350.217,172.130,49.819,159.962
C04428=1020.714,373.966,350.257,172.121,49.820,159.961
C04429=1020.705,373.719,350.297,172.112,49.820,159.960
C04430=1020.697,373.473,350.337,172.104,49.821,159.958
C04431=1020.688,373.225,350.377,172.095,49.822,159.957
C04432=1020.680,372.979,350.418,172.086,49.822,159.956
C04433=1020.671,372.733,350.458,172.077,49.823,159.955
C04434=1020.663,372.486,350.498,172.068,49.823,159.953
C04435=1020.654,372.239,350.538,172.060,49.824,159.952
C04436=1020.646,371.993,350.578,172.050,49.825,159.951
C04437=1020.637,371.747,350.618,172.042,49.825,159.950
C04438=1020.629,371.500,350.657,172.033,49.826,159.948
C04439=1020.620,371.252,350.698,172.024,49.827,159.947
C04440=1020.612,371.006,350.738,172.016,49.828,159.946
C04441=1020.604,370.759,350.778,172.007,49.829,159.945
C04442=1020.596,370.513,350.817,171.999,49.829,159.943
C04443=1020.588,370.267,350.858,171.990,49.830,159.942
C04444=1020.579,370.020,350.897,171.981,49.830,159.941
C04445=1020.571,369.773,350.937,171.972,49.831,159.940
C04446=1020.562,369.526,350.977,171.964,49.832,159.938
C04447=1020.554,369.280,351.017,171.955,49.833,159.937
C04448=1020.546,369.033,351.057,171.947,49.833,159.936
C04449=1020.538,368.786,351.096,171.938,49.835,159.935
C04450=1020.530,368.539,351.136,171.930,49.835,159.934
C04451=1020.522,368.293,351.176,171.921,49.836,159.933
C04452=1020.513,368.046,351.215,171.913,49.837,159.931
C04453=1020.505,367.799,351.254,171.905,49.838,159.930
C04454=1020.497,367.552,351.294,171.896,49.839,159.929
C04455=1020.489,367.306,351.334,171.888,49.839,159.928
C04456=1020.480,367.054,351.373,171.879,49.841,159.927
C04457=1020.473,366.803,351.413,171.870,49.842,159.926
C04458=1020.464,366.551,351.453,171.862,49.843,159.925
C04459=1020.455,366.299,351.493,171.853,49.844,159.923
C04460=1020.447,366.053,351.533,171.845,49.845,159.922
C04461=1020.439,365.806,351.571,171.836,49.846,159.921
C04462=1020.430,365.559,351.611,171.828,49.847,159.920
C04463=1020.422,365.313,351.650,171.820,49.847,159.919
C04464=1020.414,365.066,351.688,171.811,49.849,159.918
C04465=1020.406,364.819,351.727,171.804,49.850,159.917
C04466=1020.398,364.572,351.767,171.794,49.851,159.916
C04467=1020.390,364.325,351.806,171.787,49.852,159.915
C04468=1020.382,364.078,351.845,171.779,49.853,159.914
C04469=1020.374,363.832,351.884,171.770,49.854,159.912
C04470=1020.366,363.585,351.922,171.762,49.855,159.911
C04471=1020.357,363.338,351.961,171.754,49.856,159.910
C04472=1020.349,363.091,352.000,171.745,49.858,159.909
C04473=1020.342,362.844,352.039,171.738,49.859,159.908
C04474=1020.334,362.598,352.078,171.730,49.860,159.907
C04475=1020.326,362.350,352.117,171.722,49.861,159.906
C04476=1020.318,362.104,352.155,171.713,49.862,159.905
C04477=1020.310,361.857,352.194,171.705,49.863,159.904
C04478=1020.302,361.610,352.233,171.697,49.864,159.903
C04479=1020.294,361.364,352.271,171.689,49.866,159.902
C04480=1020.286,361.116,352.310,171.681,49.867,159.901
C04481=1020.278,360.869,352.349,171.673,49.868,159.900
C04482=1020.271,360.622,352.387,171.665,49.869,159.899
C04483=1020.263,360.375,352.426,171.657,49.871,159.898
C04484=1020.255,360.129,352.464,171.649,49.872,159.897
C04485=1020.247,359.882,352.503,171.641,49.873,159.896
C04486=1020.239,359.635,352.542,171.633,49.874,159.895
C04487=1020.231,359.388,352.580,171.625,49.876,159.894
C04488=1020.224,359.141,352.618,171.617,49.877,159.893
C04489=1020.216,358.894,352.656,171.609,49.879,159.892
C04490=1020.208,358.647,352.695,171.602,49.880,159.891
C04491=1020.200,358.400,352.733,171.594,49.881,159.890
C04492=1020.192,358.154,352.771,171.585,49.882,159.889
C04493=1020.184,357.906,352.809,171.578,49.884,159.888
C04494=1020.176,357.660,352.847,171.570,49.885,159.887
C04495=1020.168,357.412,352.886,171.562,49.886,159.886
C04496=1020.161,357.165,352.923,171.555,49.888,159.886
C04497=1020.153,356.918,352.962,171.546,49.890,159.885
C04498=1020.144,356.672,353.000,171.539,49.891,159.884
C04499=1020.137,356.425,353.037,171.531,49.893,159.883
C04500=1020.129,356.177,353.076,171.524,49.894,159.882
C04501=1020.122,355.930,353.113,171.516,49.895,159.881
C04502=1020.114,355.684,353.151,171.508,49.897,159.880
C04503=1020.106,355.436,353.189,171.500,49.899,159.879
C04504=1020.098,355.190,353.227,171.492,49.900,159.878
C04505=1020.091,354.943,353.264,171.484,49.902,159.877
C04506=1020.083,354.695,353.302,171.477,49.903,159.877
C04507=1020.075,354.448,353.341,171.469,49.904,159.876
C04508=1020.067,354.201,353.378,171.462,49.906,159.875
C04509=1020.060,353.955,353.416,171.454,49.908,159.874
C04510=1020.052,353.707,353.454,171.447,49.909,159.873
C04511=1020.044,353.460,353.491,171.438,49.911,159.872
C04512=1020.037,353.214,353.528,171.431,49.913,159.871
C04513=1020.029,352.969,353.566,171.424,49.915,159.871
C04514=1020.022,352.724,353.603,171.416,49.916,159.870
C04515=1020.014,352.477,353.640,171.408,49.918,159.869
C04516=1020.007,352.232,353.677,171.401,49.919,159.868
C04517=1019.999,351.986,353.714,171.394,49.921,159.867
C04518=1019.991,351.741,353.751,171.386,49.923,159.866
C04519=1019.984,351.495,353.789,171.379,49.925,159.866
C04520=1019.976,351.248,353.827,171.371,49.926,159.865
C04521=1019.968,351.001,353.864,171.364,49.928,159.864
C04522=1019.961,350.753,353.900,171.357,49.930,159.863
C04523=1019.953,350.506,353.937,171.349,49.932,159.863
C04524=1019.946,350.259,353.975,171.342,49.933,159.862
C04525=1019.938,350.012,354.012,171.334,49.935,159.861
C04526=1019.930,349.765,354.049,171.327,49.937,159.860
C04527=1019.923,349.518,354.087,171.320,49.939,159.859
C04528=1019.915,349.271,354.124,171.312,49.940,159.859
C04529=1019.908,349.024,354.161,171.305,49.942,159.858
C04530=1019.901,348.776,354.198,171.297,49.944,159.857
C04531=1019.893,348.529,354.235,171.290,49.946,159.856
C04532=1019.886,348.282,354.273,171.283,49.947,159.856
C04533=1019.878,348.035,354.309,171.275,49.949,159.855
C04534=1019.871,347.788,354.346,171.268,49.952,159.854
C04535=1019.863,347.541,354.383,171.261,49.953,159.853
C04536=1019.856,347.293,354.420,171.253,49.955,159.853
C04537=1019.848,347.046,354.457,171.246,49.957,159.852
C04538=1019.842,346.799,354.493,171.239,49.959,159.851
C04539=1019.834,346.552,354.530,171.232,49.961,159.850
C04540=1019.826,346.305,354.567,171.224,49.963,159.850
C04541=1019.819,346.058,354.604,171.217,49.965,159.849
C04542=1019.811,345.810,354.640,171.210,49.967,159.848
C04543=1019.803,345.563,354.677,171.203,49.969,159.848
C04544=1019.796,345.316,354.714,171.195,49.971,159.847
C04545=1019.789,345.069,354.750,171.188,49.973,159.846
C04546=1019.781,344.822,354.786,171.181,49.975,159.846
C04547=1019.774,344.575,354.824,171.174,49.977,159.845
C04548=1019.766,344.327,354.860,171.167,49.979,159.844
C04549=1019.759,344.080,354.896,171.160,49.982,159.844
C04550=1019.752,343.833,354.933,171.152,49.983,159.843
C04551=1019.744,343.586,354.969,171.145,49.986,159.842
C04552=1019.737,343.338,355.006,171.138,49.987,159.841
C04553=1019.730,343.091,355.042,171.131,49.990,159.841
C04554=1019.723,342.844,355.078,171.123,49.992,159.840
C04555=1019.715,342.596,355.115,171.117,49.994,159.840
C04556=1019.707,342.349,355.151,171.110,49.996,159.839
C04557=1019.701,342.102,355.187,171.103,49.998,159.838
C04558=1019.693,341.854,355.223,171.096,50.000,159.838
C04559=1019.686,341.607,355.260,171.089,50.003,159.837
C04560=1019.679,341.360,355.296,171.082,50.005,159.836
C04561=1019.672,341.112,355.332,171.074,50.007,159.836
C04562=1019.665,340.866,355.368,171.067,50.009,159.835
C04563=1019.657,340.618,355.404,171.060,50.011,159.834
C04564=1019.649,340.371,355.441,171.054,50.013,159.834
C04565=1019.643,340.124,355.477,171.047,50.016,159.833
C04566=1019.635,339.876,355.513,171.040,50.018,159.833
C04567=1019.628,339.629,355.548,171.033,50.021,159.832
C04568=1019.621,339.382,355.585,171.026,50.022,159.831
C04569=1019.614,339.135,355.620,171.019,50.025,159.831
C04570=1019.606,338.887,355.657,171.012,50.027,159.830
C04571=1019.599,338.640,355.692,171.005,50.030,159.830
C04572=1019.592,338.393,355.728,170.999,50.032,159.829
C04573=1019.585,338.146,355.764,170.992,50.034,159.829
C04574=1019.578,337.898,355.799,170.985,50.037,159.828
C04575=1019.570,337.651,355.835,170.978,50.039,159.828
C04576=1019.563,337.404,355.871,170.971,50.042,159.827
C04577=1019.556,337.157,355.906,170.964,50.044,159.826
C04578=1019.549,336.909,355.942,170.958,50.046,159.826
C04579=1019.542,336.662,355.978,170.951,50.049,159.825
C04580=1019.535,336.415,356.013,170.944,50.051,159.825
C04581=1019.527,336.167,356.049,170.937,50.054,159.824
C04582=1019.520,335.921,356.085,170.930,50.056,159.824
C04583=1019.513,335.672,356.120,170.923,50.059,159.823
C04584=1019.506,335.425,356.155,170.917,50.061,159.823
C04585=1019.499,335.178,356.191,170.910,50.063,159.822
C04586=1019.492,334.930,356.227,170.904,50.066,159.822
C04587=1019.485,334.683,356.262,170.897,50.069,159.821
C04588=1019.478,334.436,356.298,170.890,50.071,159.820
C04589=1019.471,334.189,356.333,170.884,50.074,159.820
C04590=1019.464,333.941,356.368,170.877,50.076,159.820
C04591=1019.457,333.693,356.404,170.870,50.078,159.819
C04592=1019.450,333.447,356.439,170.863,50.081,159.819
C04593=1019.443,333.199,356.475,170.856,50.084,159.818
C04594=1019.436,332.951,356.510,170.851,50.086,159.818
C04595=1019.428,332.704,356.545,170.844,50.089,159.817
C04596=1019.421,332.457,356.580,170.837,50.092,159.817
C04597=1019.415,332.209,356.615,170.830,50.094,159.816
C04598=1019.407,331.961,356.650,170.823,50.097,159.816
C04599=1019.400,331.714,356.685,170.817,50.099,159.815
C04600=1019.393,331.467,356.720,170.811,50.102,159.815
C04601=1019.386,331.220,356.755,170.804,50.105,159.814
C04602=1019.379,330.973,356.790,170.797,50.108,159.814
C04603=1019.371,330.724,356.825,170.790,50.111,159.814
C04604=1019.365,330.477,356.860,170.784,50.113,159.813
C04605=1019.358,330.230,356.895,170.778,50.116,159.813
C04606=1019.351,329.982,356.929,170.771,50.119,159.812
C04607=1019.344,329.735,356.964,170.764,50.121,159.812
C04608=1019.337,329.487,357.000,170.758,50.124,159.811
C04609=1019.330,329.240,357.035,170.752,50.127,159.811
C04610=1019.323,328.993,357.069,170.745,50.130,159.811
C04611=1019.316,328.745,357.104,170.738,50.132,159.810
C04612=1019.310,328.498,357.139,170.732,50.135,159.810
C04613=1019.302,328.250,357.173,170.726,50.138,159.809
C04614=1019.295,328.002,357.208,170.719,50.141,159.809
C04615=1019.288,327.754,357.243,170.712,50.143,159.808
C04616=1019.282,327.507,357.278,170.706,50.146,159.808
C04617=1019.275,327.260,357.312,170.700,50.149,159.808
C04618=1019.268,327.013,357.347,170.693,50.152,159.807
C04619=1019.261,326.765,357.382,170.688,50.155,159.807
C04620=1019.254,326.518,357.416,170.681,50.158,159.806
C04621=1019.247,326.270,357.451,170.674,50.161,159.806
C04622=1019.240,326.023,357.485,170.668,50.164,159.806
C04623=1019.233,325.775,357.519,170.662,50.167,159.805
C04624=1019.226,325.528,357.553,170.655,50.170,159.805
C04625=1019.219,325.280,357.588,170.649,50.173,159.805
C04626=1019.212,325.032,357.621,170.642,50.176,159.804
C04627=1019.205,324.785,357.655,170.636,50.179,159.804
C04628=1019.198,324.537,357.690,170.630,50.182,159.804
C04629=1019.191,324.290,357.724,170.623,50.185,159.803
C04630=1019.183,324.042,357.758,170.617,50.188,159.803
C04631=1019.176,323.794,357.792,170.610,50.191,159.803
C04632=1019.170,323.546,357.826,170.605,50.195,159.802
C04633=1019.163,323.300,357.861,170.598,50.198,159.802
C04634=1019.156,323.052,357.894,170.592,50.201,159.802
C04635=1019.149,322.805,357.928,170.585,50.204,159.801
C04636=1019.142,322.553,357.963,170.580,50.207,159.801
C04637=1019.135,322.302,357.997,170.573,50.210,159.801
C04638=1019.128,322.050,358.031,170.566,50.213,159.800
C04639=1019.121,321.799,358.066,170.560,50.217,159.800
C04640=1019.114,321.551,358.100,170.554,50.220,159.800
C04641=1019.108,321.304,358.134,170.548,50.222,159.799
C04642=1019.101,321.056,358.168,170.542,50.226,159.799
C04643=1019.093,320.808,358.201,170.535,50.229,159.799
C04644=1019.086,320.561,358.235,170.529,50.233,159.799
C04645=1019.080,320.314,358.269,170.523,50.236,159.798
C04646=1019.073,320.066,358.303,170.517,50.239,159.798
C04647=1019.066,319.818,358.337,170.510,50.242,159.798
C04648=1019.059,319.571,358.370,170.505,50.245,159.797
C04649=1019.053,319.323,358.405,170.498,50.249,159.797
C04650=1019.046,319.076,358.439,170.492,50.252,159.797
C04651=1019.039,318.828,358.471,170.486,50.255,159.797
C04652=1019.032,318.580,358.505,170.480,50.259,159.797
C04653=1019.026,318.332,358.540,170.473,50.262,159.796
C04654=1019.019,318.085,358.573,170.468,50.265,159.796
C04655=1019.012,317.838,358.607,170.462,50.268,159.796
C04656=1019.006,317.590,358.640,170.455,50.272,159.796
C04657=1018.999,317.342,358.674,170.450,50.274,159.795
C04658=1018.992,317.095,358.708,170.443,50.278,159.795
C04659=1018.986,316.847,358.741,170.437,50.282,159.795
C04660=1018.978,316.599,358.775,170.431,50.285,159.795
C04661=1018.972,316.352,358.808,170.425,50.288,159.794
C04662=1018.966,316.104,358.842,170.419,50.292,159.794
C04663=1018.959,315.857,358.875,170.413,50.295,159.794
C04664=1018.952,315.609,358.909,170.407,50.298,159.794
C04665=1018.946,315.361,358.942,170.401,50.302,159.793
C04666=1018.940,315.114,358.976,170.396,50.305,159.793
C04667=1018.933,314.866,359.009,170.389,50.308,159.793
C04668=1018.926,314.619,359.042,170.383,50.312,159.793
C04669=1018.919,314.370,359.075,170.377,50.315,159.793
C04670=1018.913,314.123,359.109,170.371,50.319,159.792
C04671=1018.907,313.875,359.143,170.366,50.322,159.792
C04672=1018.900,313.628,359.176,170.359,50.325,159.792
C04673=1018.894,313.380,359.209,170.353,50.329,159.792
C04674=1018.886,313.133,359.243,170.348,50.332,159.792
C04675=1018.881,312.885,359.276,170.341,50.336,159.791
C04676=1018.875,312.637,359.309,170.335,50.340,159.791
C04677=1018.867,312.389,359.343,170.330,50.343,159.791
C04678=1018.861,312.142,359.375,170.324,50.347,159.791
C04679=1018.855,311.895,359.409,170.318,50.350,159.791
C04680=1018.848,311.646,359.442,170.312,50.354,159.791
C04681=1018.842,311.399,359.475,170.305,50.357,159.790
C04682=1018.835,311.152,359.509,170.300,50.360,159.790
C04683=1018.829,310.904,359.541,170.294,50.364,159.790
C04684=1018.823,310.656,359.575,170.289,50.367,159.790
C04685=1018.817,310.408,359.608,170.282,50.371,159.790
C04686=1018.810,310.161,359.641,170.277,50.374,159.789
C04687=1018.804,309.913,359.674,170.271,50.378,159.789
C04688=1018.797,309.665,359.707,170.265,50.382,159.789
C04689=1018.791,309.417,359.740,170.260,50.386,159.789
C04690=1018.784,309.170,359.772,170.253,50.390,159.789
C04691=1018.777,308.923,359.805,170.248,50.394,159.789
C04692=1018.770,308.675,359.837,170.242,50.397,159.789
C04693=1018.764,308.429,359.869,170.236,50.401,159.789
C04694=1018.757,308.182,359.902,170.230,50.405,159.789
C04695=1018.750,307.935,359.934,170.225,50.409,159.788
C04696=1018.744,307.688,359.966,170.219,50.412,159.788
C04697=1018.737,307.441,359.998,170.213,50.417,159.788
C04698=1018.730,307.195,360.031,170.208,50.420,159.788
C04699=1018.724,306.948,360.063,170.201,50.424,159.788
C04700=1018.717,306.700,360.096,170.195,50.428,159.788
C04701=1018.711,306.452,360.128,170.190,50.431,159.788
C04702=1018.704,306.204,360.160,170.184,50.436,159.788
C04703=1018.697,305.957,360.193,170.178,50.440,159.788
C04704=1018.691,305.709,360.225,170.173,50.444,159.788
C04705=1018.684,305.461,360.257,170.167,50.447,159.788
C04706=1018.677,305.213,360.290,170.161,50.452,159.788
C04707=1018.671,304.965,360.321,170.156,50.455,159.787
C04708=1018.664,304.718,360.354,170.150,50.459,159.787
C04709=1018.657,304.470,360.386,170.144,50.463,159.787
C04710=1018.651,304.222,360.418,170.139,50.467,159.787
C04711=1018.645,303.974,360.451,170.133,50.471,159.787
C04712=1018.638,303.727,360.482,170.127,50.475,159.787
C04713=1018.632,303.479,360.515,170.122,50.479,159.787
C04714=1018.625,303.231,360.547,170.116,50.483,159.787
C04715=1018.619,302.983,360.579,170.110,50.487,159.787
C04716=1018.612,302.736,360.611,170.105,50.491,159.787
C04717=1018.606,302.488,360.643,170.099,50.495,159.787
C04718=1018.600,302.240,360.675,170.093,50.499,159.787
C04719=1018.593,301.992,360.708,170.088,50.503,159.787
C04720=1018.587,301.744,360.740,170.082,50.508,159.787
C04721=1018.580,301.496,360.771,170.077,50.511,159.787
C04722=1018.574,301.249,360.804,170.071,50.515,159.787
C04723=1018.567,301.001,360.835,170.065,50.520,159.787
C04724=1018.561,300.753,360.867,170.060,50.524,159.787
C04725=1018.555,300.505,360.900,170.054,50.527,159.787
C04726=1018.548,300.257,360.931,170.048,50.532,159.787
C04727=1018.542,300.009,360.963,170.043,50.536,159.787
C04728=1018.535,299.762,360.996,170.037,50.540,159.787
C04729=1018.529,299.513,361.028,170.032,50.544,159.787
C04730=1018.523,299.266,361.059,170.026,50.548,159.787
C04731=1018.517,299.018,361.091,170.020,50.552,159.787
C04732=1018.511,298.770,361.123,170.015,50.556,159.787
C04733=1018.504,298.523,361.155,170.009,50.561,159.787
C04734=1018.498,298.274,361.187,170.004,50.565,159.787
C04735=1018.491,298.026,361.218,169.999,50.569,159.787
C04736=1018.485,297.778,361.250,169.993,50.574,159.787
C04737=1018.479,297.531,361.281,169.988,50.578,159.787
C04738=1018.473,297.283,361.314,169.982,50.582,159.787
C04739=1018.466,297.035,361.346,169.976,50.586,159.787
C04740=1018.460,296.787,361.378,169.971,50.590,159.787
C04741=1018.454,296.539,361.410,169.966,50.595,159.787
C04742=1018.448,296.292,361.441,169.961,50.599,159.787
C04743=1018.442,296.044,361.473,169.955,50.603,159.787
C04744=1018.436,295.796,361.504,169.950,50.607,159.787
C04745=1018.430,295.548,361.536,169.944,50.612,159.787
C04746=1018.423,295.300,361.567,169.938,50.616,159.787
C04747=1018.417,295.052,361.599,169.933,50.620,159.787
C04748=1018.411,294.804,361.631,169.927,50.624,159.787
C04749=1018.405,294.557,361.662,169.923,50.628,159.787
C04750=1018.399,294.308,361.694,169.917,50.633,159.787
C04751=1018.393,294.061,361.726,169.911,50.637,159.787
C04752=1018.387,293.822,361.756,169.906,50.641,159.787
C04753=1018.381,293.584,361.786,169.901,50.645,159.787
C04754=1018.376,293.346,361.817,169.895,50.650,159.787
C04755=1018.370,293.108,361.847,169.890,50.654,159.788
C04756=1018.363,292.870,361.877,169.886,50.658,159.788
C04757=1018.358,292.632,361.907,169.880,50.663,159.788
C04758=1018.351,292.394,361.937,169.875,50.667,159.788
C04759=1018.346,292.156,361.967,169.870,50.671,159.788
C04760=1018.340,291.909,361.998,169.864,50.675,159.788
C04761=1018.333,291.661,362.029,169.859,50.680,159.788
C04762=1018.326,291.413,362.060,169.854,50.684,159.788
C04763=1018.320,291.165,362.091,169.849,50.689,159.788
C04764=1018.314,290.917,362.122,169.843,50.694,159.788
C04765=1018.308,290.669,362.154,169.838,50.698,159.788
C04766=1018.302,290.421,362.184,169.832,50.703,159.789
C04767=1018.295,290.173,362.216,169.827,50.707,159.789
C04768=1018.289,289.925,362.246,169.822,50.712,159.789
C04769=1018.283,289.677,362.278,169.816,50.716,159.789
C04770=1018.277,289.429,362.308,169.812,50.721,159.789
C04771=1018.271,289.181,362.339,169.806,50.725,159.789
C04772=1018.264,288.933,362.370,169.800,50.730,159.789
C04773=1018.258,288.685,362.400,169.796,50.735,159.790
C04774=1018.251,288.437,362.432,169.790,50.740,159.790
C04775=1018.245,288.189,362.462,169.785,50.745,159.790
C04776=1018.239,287.941,362.493,169.780,50.749,159.790
C04777=1018.233,287.694,362.524,169.774,50.754,159.790
C04778=1018.226,287.445,362.555,169.769,50.759,159.790
C04779=1018.221,287.197,362.585,169.764,50.763,159.790
C04780=1018.214,286.949,362.617,169.759,50.768,159.791
C04781=1018.208,286.702,362.647,169.753,50.773,159.791
C04782=1018.202,286.453,362.678,169.748,50.777,159.791
C04783=1018.196,286.205,362.708,169.743,50.782,159.791
C04784=1018.189,285.957,362.739,169.737,50.787,159.791
C04785=1018.183,285.710,362.770,169.733,50.792,159.792
C04786=1018.177,285.461,362.800,169.727,50.796,159.792
C04787=1018.171,285.213,362.831,169.722,50.801,159.792
C04788=1018.165,284.965,362.861,169.717,50.806,159.792
C04789=1018.159,284.717,362.892,169.712,50.811,159.792
C04790=1018.153,284.469,362.922,169.706,50.816,159.792
C04791=1018.147,284.221,362.953,169.701,50.820,159.792
C04792=1018.141,283.973,362.983,169.696,50.825,159.793
C04793=1018.134,283.725,363.013,169.690,50.830,159.793
C04794=1018.128,283.477,363.044,169.686,50.835,159.793
C04795=1018.122,283.229,363.074,169.680,50.840,159.793
C04796=1018.116,282.980,363.105,169.675,50.845,159.794
C04797=1018.109,282.733,363.135,169.670,50.850,159.794
C04798=1018.103,282.485,363.165,169.665,50.855,159.794
C04799=1018.097,282.236,363.196,169.660,50.860,159.794
C04800=1018.091,281.989,363.226,169.654,50.865,159.794
C04801=1018.084,281.741,363.256,169.650,50.870,159.795
C04802=1018.078,281.492,363.286,169.644,50.875,159.795
C04803=1018.073,281.244,363.316,169.639,50.880,159.795
C04804=1018.067,280.996,363.346,169.634,50.885,159.795
C04805=1018.060,280.748,363.377,169.629,50.890,159.796
C04806=1018.054,280.500,363.407,169.624,50.896,159.796
C04807=1018.048,280.252,363.437,169.619,50.900,159.796
C04808=1018.042,280.003,363.467,169.614,50.905,159.796
C04809=1018.035,279.756,363.497,169.608,50.911,159.797
C04810=1018.029,279.508,363.527,169.603,50.916,159.797
C04811=1018.024,279.260,363.557,169.599,50.920,159.797
C04812=1018.018,279.028,363.586,169.594,50.925,159.797
C04813=1018.012,278.796,363.613,169.589,50.930,159.798
C04814=1018.006,278.563,363.641,169.584,50.935,159.798
C04815=1018.001,278.332,363.670,169.580,50.940,159.798
C04816=1017.996,278.100,363.698,169.575,50.944,159.798
C04817=1017.989,277.868,363.726,169.570,50.949,159.799
C04818=1017.984,277.637,363.754,169.565,50.954,159.799
C04819=1017.978,277.405,363.782,169.561,50.959,159.799
C04820=1017.973,277.156,363.812,169.555,50.964,159.799
C04821=1017.966,276.909,363.841,169.550,50.969,159.799
C04822=1017.960,276.660,363.872,169.546,50.974,159.800
C04823=1017.955,276.412,363.902,169.541,50.980,159.800
C04824=1017.948,276.164,363.932,169.535,50.985,159.800
C04825=1017.942,275.916,363.961,169.531,50.989,159.801
C04826=1017.936,275.668,363.990,169.526,50.995,159.801
C04827=1017.930,275.420,364.021,169.520,51.000,159.801
C04828=1017.924,275.171,364.050,169.515,51.006,159.802
C04829=1017.918,274.923,364.080,169.511,51.011,159.802
C04830=1017.911,274.675,364.109,169.506,51.017,159.802
C04831=1017.906,274.427,364.139,169.500,51.022,159.802
C04832=1017.899,274.179,364.169,169.495,51.027,159.803
C04833=1017.894,273.931,364.198,169.491,51.032,159.803
C04834=1017.888,273.682,364.227,169.486,51.038,159.803
C04835=1017.882,273.435,364.258,169.480,51.043,159.804
C04836=1017.876,273.187,364.287,169.475,51.049,159.804
C04837=1017.869,272.937,364.317,169.471,51.054,159.804
C04838=1017.863,272.689,364.346,169.466,51.059,159.805
C04839=1017.857,272.441,364.376,169.460,51.065,159.805
C04840=1017.851,272.193,364.405,169.456,51.070,159.805
C04841=1017.846,271.945,364.435,169.451,51.076,159.806
C04842=1017.839,271.697,364.464,169.446,51.081,159.806
C04843=1017.833,271.449,364.493,169.441,51.087,159.806
C04844=1017.827,271.201,364.523,169.436,51.092,159.807
C04845=1017.821,270.953,364.552,169.431,51.097,159.807
C04846=1017.816,270.704,364.582,169.426,51.103,159.807
C04847=1017.809,270.456,364.611,169.421,51.109,159.808
C04848=1017.803,270.208,364.640,169.416,51.114,159.808
C04849=1017.798,269.959,364.670,169.412,51.119,159.808
C04850=1017.791,269.711,364.699,169.407,51.125,159.809
C04851=1017.786,269.463,364.728,169.401,51.131,159.809
C04852=1017.780,269.215,364.757,169.396,51.136,159.809
C04853=1017.773,268.967,364.787,169.392,51.141,159.810
C04854=1017.767,268.719,364.816,169.387,51.147,159.810
C04855=1017.762,268.471,364.845,169.382,51.153,159.811
C04856=1017.756,268.223,364.874,169.377,51.159,159.811
C04857=1017.750,267.975,364.903,169.372,51.164,159.811
C04858=1017.743,267.726,364.932,169.368,51.170,159.812
C04859=1017.738,267.478,364.962,169.362,51.175,159.812
C04860=1017.732,267.229,364.990,169.357,51.181,159.813
C04861=1017.726,266.981,365.019,169.352,51.187,159.813
C04862=1017.719,266.733,365.048,169.347,51.192,159.813
C04863=1017.714,266.484,365.078,169.343,51.198,159.814
C04864=1017.708,266.236,365.107,169.338,51.204,159.814
C04865=1017.701,265.988,365.136,169.333,51.209,159.815
C04866=1017.696,265.740,365.164,169.328,51.215,159.815
C04867=1017.690,265.492,365.193,169.323,51.221,159.815
C04868=1017.684,265.244,365.222,169.319,51.226,159.816
C04869=1017.678,264.995,365.251,169.314,51.232,159.816
C04870=1017.672,264.747,365.280,169.309,51.238,159.817
C04871=1017.666,264.499,365.309,169.304,51.244,159.817
C04872=1017.660,264.270,365.335,169.300,51.249,159.817
C04873=1017.655,264.039,365.361,169.296,51.255,159.818
C04874=1017.649,263.810,365.388,169.291,51.261,159.818
C04875=1017.644,263.580,365.415,169.287,51.266,159.819
C04876=1017.638,263.351,365.441,169.283,51.271,159.819
C04877=1017.632,263.121,365.468,169.277,51.277,159.819
C04878=1017.627,262.891,365.494,169.273,51.282,159.820
C04879=1017.622,262.662,365.521,169.269,51.288,159.820
C04880=1017.616,262.413,365.549,169.264,51.293,159.821
C04881=1017.610,262.165,365.578,169.259,51.299,159.821
C04882=1017.604,261.917,365.607,169.254,51.305,159.822
C04883=1017.598,261.668,365.636,169.250,51.311,159.822
C04884=1017.593,261.420,365.664,169.245,51.317,159.823
C04885=1017.586,261.172,365.693,169.241,51.323,159.823
C04886=1017.580,260.923,365.721,169.236,51.329,159.823
C04887=1017.575,260.676,365.750,169.231,51.335,159.824
C04888=1017.569,260.427,365.778,169.226,51.341,159.824
C04889=1017.563,260.179,365.807,169.221,51.347,159.825
C04890=1017.557,259.930,365.836,169.216,51.353,159.825
C04891=1017.551,259.682,365.863,169.211,51.359,159.826
C04892=1017.545,259.434,365.893,169.207,51.365,159.826
C04893=1017.538,259.186,365.920,169.202,51.371,159.827
C04894=1017.533,258.938,365.948,169.198,51.377,159.827
C04895=1017.527,258.689,365.977,169.193,51.383,159.828
C04896=1017.520,258.441,366.004,169.189,51.390,159.828
C04897=1017.514,258.192,366.033,169.184,51.396,159.829
C04898=1017.509,257.944,366.061,169.179,51.402,159.829
C04899=1017.502,257.696,366.089,169.174,51.408,159.830
C04900=1017.496,257.447,366.117,169.169,51.414,159.830
C04901=1017.490,257.199,366.145,169.165,51.421,159.831
C04902=1017.484,256.951,366.173,169.160,51.427,159.831
C04903=1017.478,256.702,366.201,169.155,51.433,159.832
C04904=1017.472,256.454,366.229,169.151,51.440,159.833
C04905=1017.466,256.205,366.257,169.146,51.446,159.833
C04906=1017.460,255.957,366.285,169.141,51.452,159.833
C04907=1017.454,255.709,366.313,169.136,51.459,159.834
C04908=1017.448,255.460,366.341,169.131,51.464,159.834
C04909=1017.443,255.212,366.369,169.127,51.471,159.835
C04910=1017.436,254.964,366.397,169.122,51.477,159.836
C04911=1017.430,254.715,366.425,169.118,51.484,159.836
C04912=1017.424,254.467,366.452,169.113,51.490,159.837
C04913=1017.418,254.218,366.481,169.108,51.496,159.837
C04914=1017.413,253.970,366.509,169.103,51.503,159.838
C04915=1017.406,253.722,366.536,169.099,51.509,159.838
C04916=1017.400,253.473,366.565,169.094,51.515,159.839
C04917=1017.395,253.225,366.593,169.089,51.522,159.839
C04918=1017.388,252.977,366.620,169.085,51.528,159.840
C04919=1017.383,252.728,366.648,169.080,51.535,159.841
C04920=1017.377,252.480,366.675,169.075,51.541,159.841
C04921=1017.371,252.232,366.703,169.071,51.548,159.842
C04922=1017.365,251.983,366.732,169.066,51.554,159.842
C04923=1017.359,251.735,366.759,169.061,51.560,159.843
C04924=1017.353,251.486,366.787,169.057,51.567,159.843
C04925=1017.348,251.238,366.815,169.052,51.573,159.844
C04926=1017.342,250.989,366.842,169.049,51.579,159.845
C04927=1017.336,250.741,366.870,169.044,51.586,159.845
C04928=1017.330,250.492,366.899,169.039,51.592,159.846
C04929=1017.324,250.245,366.926,169.035,51.599,159.846
C04930=1017.319,249.996,366.953,169.030,51.606,159.847
C04931=1017.312,249.748,366.981,169.026,51.612,159.848
C04932=1017.307,249.517,367.006,169.021,51.618,159.848
C04933=1017.302,249.287,367.033,169.017,51.624,159.849
C04934=1017.297,249.056,367.058,169.012,51.630,159.849
C04935=1017.291,248.825,367.084,169.009,51.636,159.850
C04936=1017.286,248.595,367.110,169.004,51.642,159.850
C04937=1017.281,248.364,367.135,169.000,51.648,159.851
C04938=1017.276,248.135,367.161,168.995,51.655,159.851
C04939=1017.270,247.904,367.186,168.991,51.660,159.852
C04940=1017.264,247.655,367.215,168.987,51.667,159.852
C04941=1017.258,247.407,367.241,168.982,51.673,159.853
C04942=1017.253,247.159,367.269,168.978,51.680,159.854
C04943=1017.246,246.910,367.297,168.974,51.687,159.854
C04944=1017.241,246.661,367.324,168.969,51.694,159.855
C04945=1017.236,246.413,367.352,168.964,51.700,159.856
C04946=1017.230,246.164,367.379,168.960,51.707,159.856
C04947=1017.224,245.916,367.407,168.955,51.713,159.857
C04948=1017.218,245.669,367.435,168.951,51.720,159.857
C04949=1017.213,245.419,367.462,168.946,51.726,159.858
C04950=1017.207,245.171,367.490,168.942,51.734,159.859
C04951=1017.201,244.923,367.517,168.937,51.740,159.859
C04952=1017.196,244.675,367.545,168.932,51.747,159.860
C04953=1017.190,244.425,367.572,168.927,51.754,159.860
C04954=1017.184,244.178,367.600,168.923,51.760,159.861
C04955=1017.179,243.929,367.627,168.919,51.768,159.862
C04956=1017.174,243.681,367.654,168.914,51.774,159.862
C04957=1017.168,243.432,367.682,168.909,51.781,159.863
C04958=1017.163,243.183,367.709,168.905,51.787,159.863
C04959=1017.156,242.935,367.737,168.901,51.794,159.864
C04960=1017.151,242.687,367.763,168.896,51.801,159.865
C04961=1017.145,242.438,367.791,168.892,51.808,159.865
C04962=1017.139,242.190,367.818,168.888,51.815,159.866
C04963=1017.133,241.942,367.845,168.883,51.821,159.867
C04964=1017.128,241.693,367.872,168.879,51.829,159.868
C04965=1017.122,241.444,367.899,168.874,51.835,159.868
C04966=1017.116,241.196,367.926,168.869,51.843,159.869
C04967=1017.111,240.947,367.954,168.865,51.849,159.870
C04968=1017.105,240.699,367.980,168.861,51.857,159.870
C04969=1017.099,240.451,368.007,168.856,51.863,159.871
C04970=1017.093,240.201,368.035,168.852,51.871,159.872
C04971=1017.088,239.953,368.061,168.847,51.877,159.872
C04972=1017.082,239.705,368.089,168.843,51.884,159.873
C04973=1017.077,239.457,368.116,168.839,51.891,159.874
C04974=1017.071,239.208,368.142,168.834,51.899,159.874
C04975=1017.064,238.959,368.169,168.829,51.905,159.875
C04976=1017.059,238.711,368.196,168.825,51.912,159.876
C04977=1017.053,238.462,368.223,168.821,51.920,159.877
C04978=1017.047,238.214,368.249,168.816,51.926,159.877
C04979=1017.041,237.966,368.276,168.812,51.934,159.878
C04980=1017.036,237.717,368.303,168.807,51.941,159.879
C04981=1017.031,237.469,368.330,168.803,51.948,159.879
C04982=1017.025,237.220,368.357,168.798,51.955,159.880
C04983=1017.018,236.971,368.384,168.794,51.962,159.881
C04984=1017.013,236.723,368.410,168.789,51.970,159.882
C04985=1017.007,236.475,368.437,168.785,51.977,159.882
C04986=1017.001,236.226,368.464,168.780,51.984,159.883
C04987=1016.996,235.977,368.489,168.776,51.991,159.884
C04988=1016.990,235.729,368.516,168.772,51.998,159.885
C04989=1016.984,235.481,368.543,168.767,52.006,159.885
C04990=1016.978,235.232,368.569,168.763,52.013,159.886
C04991=1016.973,234.984,368.596,168.759,52.021,159.887
C04992=1016.967,234.750,368.620,168.754,52.027,159.887
C04993=1016.961,234.516,368.645,168.750,52.034,159.888
C04994=1016.956,234.282,368.671,168.746,52.041,159.889
C04995=1016.951,234.049,368.695,168.742,52.048,159.890
C04996=1016.945,233.815,368.721,168.738,52.055,159.890
C04997=1016.940,233.580,368.745,168.734,52.062,159.891
C04998=1016.934,233.347,368.770,168.730,52.068,159.892
C04999=1016.929,233.113,368.795,168.725,52.076,159.892
C05000=1016.923,232.864,368.822,168.721,52.083,159.893
C05001=1016.918,232.615,368.848,168.717,52.090,159.894
C05002=1016.912,232.367,368.875,168.712,52.098,159.895
C05003=1016.906,232.119,368.901,168.708,52.105,159.896
C05004=1016.901,231.870,368.927,168.704,52.113,159.896
C05005=1016.895,231.621,368.954,168.699,52.120,159.897
C05006=1016.889,231.372,368.980,168.695,52.128,159.898
C05007=1016.884,231.124,369.006,168.691,52.135,159.899
C05008=1016.878,230.876,369.033,168.687,52.142,159.899
C05009=1016.873,230.627,369.059,168.682,52.150,159.900
C05010=1016.867,230.379,369.085,168.677,52.157,159.901
C05011=1016.861,230.131,369.112,168.673,52.164,159.902
C05012=1016.856,229.882,369.138,168.669,52.173,159.903
C05013=1016.849,229.634,369.164,168.665,52.180,159.903
C05014=1016.844,229.385,369.190,168.661,52.187,159.904
C05015=1016.838,229.136,369.217,168.655,52.195,159.905
C05016=1016.833,228.887,369.242,168.651,52.202,159.906
C05017=1016.827,228.639,369.269,168.648,52.210,159.907
C05018=1016.821,228.390,369.294,168.643,52.218,159.907
C05019=1016.815,228.141,369.320,168.639,52.225,159.908
C05020=1016.810,227.894,369.347,168.634,52.233,159.909
C05021=1016.805,227.645,369.373,168.630,52.241,159.910
C05022=1016.799,227.396,369.399,168.626,52.248,159.911
C05023=1016.793,227.147,369.425,168.621,52.256,159.911
C05024=1016.787,226.899,369.450,168.617,52.264,159.913
C05025=1016.781,226.650,369.477,168.613,52.271,159.913
C05026=1016.776,226.401,369.503,168.608,52.279,159.914
C05027=1016.770,226.153,369.530,168.604,52.287,159.915
C05028=1016.764,225.905,369.555,168.599,52.295,159.916
C05029=1016.759,225.656,369.581,168.596,52.303,159.917
C05030=1016.753,225.407,369.606,168.591,52.311,159.917
C05031=1016.747,225.158,369.632,168.587,52.319,159.918
C05032=1016.741,224.910,369.658,168.582,52.326,159.919
C05033=1016.735,224.661,369.684,168.578,52.334,159.920
C05034=1016.730,224.413,369.709,168.573,52.342,159.921
C05035=1016.724,224.164,369.735,168.570,52.350,159.922
C05036=1016.719,223.915,369.761,168.566,52.357,159.923
C05037=1016.713,223.667,369.786,168.561,52.366,159.924
C05038=1016.707,223.418,369.812,168.557,52.374,159.925
C05039=1016.701,223.170,369.838,168.552,52.382,159.925
C05040=1016.696,222.921,369.864,168.549,52.390,159.926
C05041=1016.690,222.673,369.889,168.544,52.397,159.927
C05042=1016.684,222.424,369.915,168.540,52.405,159.928
C05043=1016.679,222.175,369.941,168.535,52.414,159.929
C05044=1016.673,221.927,369.966,168.531,52.421,159.930
C05045=1016.668,221.678,369.992,168.527,52.429,159.931
C05046=1016.661,221.429,370.017,168.523,52.438,159.932
C05047=1016.656,221.180,370.043,168.518,52.445,159.932
C05048=1016.650,220.932,370.068,168.513,52.454,159.933
C05049=1016.645,220.683,370.094,168.510,52.462,159.934
C05050=1016.639,220.435,370.119,168.505,52.469,159.935
C05051=1016.633,220.186,370.145,168.501,52.477,159.936
C05052=1016.628,219.948,370.170,168.498,52.486,159.937
C05053=1016.622,219.710,370.194,168.493,52.493,159.938
C05054=1016.617,219.473,370.219,168.489,52.501,159.939
C05055=1016.612,219.234,370.243,168.485,52.509,159.940
C05056=1016.607,218.996,370.267,168.481,52.516,159.940
C05057=1016.601,218.758,370.292,168.477,52.524,159.941
C05058=1016.596,218.521,370.316,168.472,52.532,159.942
C05059=1016.591,218.282,370.340,168.469,52.540,159.943
C05060=1016.585,218.033,370.366,168.465,52.548,159.944
C05061=1016.580,217.785,370.391,168.460,52.556,159.945
C05062=1016.574,217.536,370.417,168.456,52.564,159.946
C05063=1016.568,217.288,370.442,168.452,52.572,159.947
C05064=1016.562,217.039,370.467,168.447,52.581,159.948
C05065=1016.556,216.790,370.492,168.443,52.589,159.949
C05066=1016.551,216.542,370.517,168.439,52.597,159.950
C05067=1016.545,216.293,370.542,168.435,52.606,159.951
C05068=1016.539,216.044,370.567,168.430,52.615,159.952
C05069=1016.534,215.796,370.593,168.427,52.623,159.953
C05070=1016.528,215.547,370.618,168.422,52.631,159.954
C05071=1016.523,215.298,370.642,168.418,52.640,159.955
C05072=1016.516,215.050,370.668,168.414,52.648,159.956
C05073=1016.511,214.801,370.694,168.410,52.656,159.956
C05074=1016.506,214.552,370.718,168.405,52.665,159.957
C05075=1016.499,214.304,370.743,168.401,52.673,159.958
C05076=1016.494,214.056,370.768,168.397,52.681,159.959
C05077=1016.489,213.806,370.793,168.393,52.690,159.960
C05078=1016.483,213.558,370.818,168.388,52.699,159.961
C05079=1016.477,213.309,370.843,168.385,52.707,159.962
C05080=1016.471,213.060,370.868,168.380,52.715,159.963
C05081=1016.466,212.812,370.894,168.376,52.724,159.964
C05082=1016.460,212.562,370.918,168.372,52.732,159.965
C05083=1016.454,212.314,370.943,168.368,52.741,159.966
C05084=1016.449,212.065,370.968,168.363,52.749,159.967
C05085=1016.444,211.817,370.994,168.359,52.758,159.968
C05086=1016.438,211.568,371.018,168.355,52.766,159.969
C05087=1016.432,211.320,371.043,168.351,52.775,159.970
C05088=1016.426,211.070,371.068,168.347,52.784,159.971
C05089=1016.421,210.822,371.093,168.343,52.792,159.972
C05090=1016.416,210.573,371.118,168.339,52.801,159.973
C05091=1016.410,210.325,371.143,168.334,52.809,159.974
C05092=1016.404,210.076,371.168,168.330,52.818,159.975
C05093=1016.398,209.828,371.193,168.326,52.826,159.976
C05094=1016.393,209.578,371.218,168.322,52.835,159.977
C05095=1016.388,209.330,371.243,168.318,52.844,159.978
C05096=1016.382,209.081,371.267,168.314,52.853,159.980
C05097=1016.376,208.832,371.292,168.309,52.861,159.980
C05098=1016.371,208.584,371.317,168.305,52.871,159.982
C05099=1016.365,208.335,371.341,168.301,52.879,159.983
C05100=1016.360,208.086,371.365,168.297,52.888,159.984
C05101=1016.354,207.837,371.390,168.293,52.896,159.985
C05102=1016.348,207.589,371.415,168.289,52.905,159.986
C05103=1016.342,207.340,371.440,168.284,52.914,159.987
C05104=1016.337,207.091,371.464,168.280,52.923,159.988
C05105=1016.332,206.843,371.488,168.276,52.932,159.989
C05106=1016.325,206.594,371.514,168.273,52.941,159.990
C05107=1016.320,206.345,371.538,168.269,52.950,159.991
C05108=1016.315,206.097,371.562,168.264,52.958,159.992
C05109=1016.309,205.847,371.587,168.260,52.967,159.993
C05110=1016.304,205.599,371.611,168.256,52.977,159.994
C05111=1016.297,205.350,371.636,168.251,52.985,159.995
C05112=1016.292,205.112,371.659,168.247,52.994,159.996
C05113=1016.287,204.874,371.683,168.244,53.002,159.997
C05114=1016.282,204.637,371.706,168.239,53.011,159.998
C05115=1016.276,204.399,371.729,168.236,53.020,160.000
C05116=1016.271,204.161,371.752,168.232,53.028,160.001
C05117=1016.266,203.923,371.776,168.227,53.037,160.001
C05118=1016.260,203.684,371.799,168.224,53.046,160.003
C05119=1016.254,203.447,371.822,168.220,53.054,160.004
C05120=1016.236,202.432,371.914,167.720,52.980,159.885
C05121=1016.231,202.182,371.937,167.715,52.990,159.886
C05122=1016.226,201.934,371.960,167.711,53.000,159.887
C05123=1016.222,201.685,371.982,167.706,53.011,159.889
C05124=1016.217,201.437,372.005,167.701,53.021,159.890
C05125=1016.213,201.187,372.028,167.696,53.031,159.891
C05126=1016.208,200.938,372.050,167.692,53.042,159.892
C05127=1016.203,200.689,372.073,167.688,53.052,159.893
C05128=1016.199,200.440,372.096,167.683,53.062,159.895
C05129=1016.194,200.192,372.118,167.679,53.072,159.896
C05130=1016.189,199.942,372.141,167.674,53.082,159.897
C05131=1016.185,199.693,372.164,167.669,53.093,159.898
C05132=1016.180,199.445,372.186,167.664,53.102,159.899
C05133=1016.176,199.196,372.209,167.659,53.113,159.900
C05134=1016.171,198.947,372.230,167.655,53.123,159.901
C05135=1016.167,198.697,372.253,167.651,53.134,159.903
C05136=1016.162,198.448,372.275,167.646,53.145,159.904
C05137=1016.157,198.199,372.297,167.641,53.155,159.905
C05138=1016.153,197.951,372.320,167.636,53.165,159.906
C05139=1016.148,197.702,372.342,167.632,53.176,159.908
C05140=1016.142,197.453,372.364,167.627,53.186,159.909
C05141=1016.138,197.204,372.387,167.622,53.196,159.910
C05142=1016.133,196.955,372.409,167.618,53.207,159.911
C05143=1016.129,196.706,372.431,167.613,53.217,159.912
C05144=1016.124,196.457,372.452,167.609,53.228,159.914
C05145=1016.120,196.208,372.475,167.604,53.238,159.915
C05146=1016.115,195.959,372.497,167.600,53.249,159.916
C05147=1016.110,195.710,372.519,167.595,53.259,159.917
C05148=1016.105,195.460,372.541,167.590,53.269,159.918
C05149=1016.101,195.212,372.563,167.586,53.280,159.920
C05150=1016.096,194.963,372.585,167.581,53.290,159.921
C05151=1016.092,194.714,372.608,167.577,53.300,159.922
C05152=1016.087,194.465,372.629,167.573,53.311,159.923
C05153=1016.082,194.216,372.651,167.569,53.322,159.925
C05154=1016.077,193.967,372.673,167.564,53.332,159.926
C05155=1016.073,193.718,372.696,167.559,53.342,159.927
C05156=1016.068,193.469,372.717,167.555,53.353,159.928
C05157=1016.064,193.220,372.739,167.550,53.363,159.929
C05158=1016.060,192.971,372.761,167.545,53.374,159.930
C05159=1016.055,192.722,372.783,167.541,53.384,159.932
C05160=1016.050,192.473,372.805,167.536,53.394,159.933
C05161=1016.045,192.224,372.827,167.533,53.404,159.934
C05162=1016.041,191.975,372.849,167.528,53.416,159.936
C05163=1016.036,191.726,372.871,167.524,53.426,159.937
C05164=1016.031,191.478,372.893,167.519,53.436,159.938
C05165=1016.027,191.228,372.914,167.515,53.447,159.939
C05166=1016.023,190.979,372.936,167.510,53.457,159.940
C05167=1016.018,190.730,372.958,167.505,53.468,159.941
C05168=1016.013,190.481,372.980,167.502,53.478,159.943
C05169=1016.009,190.232,373.003,167.497,53.488,159.944
C05170=1016.005,189.983,373.024,167.493,53.498,159.945
C05171=1016.000,189.734,373.046,167.489,53.510,159.946
C05172=1015.995,189.485,373.068,167.484,53.520,159.948
C05173=1015.991,189.236,373.090,167.479,53.530,159.949
C05174=1015.986,188.987,373.111,167.476,53.540,159.950
C05175=1015.982,188.738,373.133,167.471,53.551,159.951
C05176=1015.977,188.489,373.155,167.467,53.561,159.952
C05177=1015.973,188.241,373.177,167.462,53.572,159.954
C05178=1015.969,187.991,373.198,167.457,53.582,159.955
C05179=1015.964,187.742,373.220,167.454,53.592,159.956
C05180=1015.960,187.493,373.242,167.449,53.603,159.957
C05181=1015.955,187.213,373.266,167.445,53.615,159.959
C05182=1015.949,186.933,373.291,167.440,53.626,159.960
C05183=1015.944,186.653,373.315,167.435,53.639,159.962
C05184=1015.940,186.373,373.340,167.431,53.650,159.963
C05185=1015.935,186.124,373.362,167.426,53.660,159.964
C05186=1015.931,185.875,373.383,167.422,53.671,159.965
C05187=1015.926,185.626,373.405,167.417,53.681,159.967
C05188=1015.922,185.378,373.427,167.414,53.691,159.968
C05189=1015.918,185.128,373.448,167.409,53.702,159.969
C05190=1015.913,184.879,373.470,167.404,53.712,159.970
C05191=1015.908,184.630,373.491,167.401,53.722,159.972
C05192=1015.904,184.381,373.514,167.397,53.733,159.973
C05193=1015.900,184.132,373.534,167.392,53.744,159.974
C05194=1015.896,183.883,373.556,167.388,53.754,159.975
C05195=1015.891,183.634,373.579,167.384,53.764,159.977
C05196=1015.887,183.385,373.600,167.380,53.775,159.978
C05197=1015.883,183.136,373.621,167.375,53.785,159.979
C05198=1015.878,182.887,373.642,167.372,53.795,159.980
C05199=1015.874,182.638,373.665,167.367,53.806,159.981
C05200=1015.870,182.388,373.686,167.363,53.816,159.983
C05201=1015.865,182.140,373.708,167.359,53.827,159.984
C05202=1015.861,181.891,373.729,167.355,53.837,159.985
C05203=1015.857,181.641,373.750,167.350,53.848,159.986
C05204=1015.852,181.392,373.771,167.347,53.858,159.988
C05205=1015.847,181.143,373.793,167.343,53.869,159.989
C05206=1015.842,180.894,373.814,167.339,53.880,159.991
C05207=1015.838,180.645,373.834,167.334,53.891,159.992
C05208=1015.833,180.396,373.855,167.330,53.902,159.993
C05209=1015.828,180.147,373.876,167.326,53.912,159.994
C05210=1015.824,179.897,373.897,167.321,53.923,159.995
C05211=1015.820,179.649,373.918,167.318,53.934,159.997
C05212=1015.814,179.400,373.938,167.314,53.944,159.998
C05213=1015.810,179.150,373.960,167.310,53.955,160.000
C05214=1015.805,178.901,373.980,167.305,53.966,160.001
C05215=1015.800,178.653,374.002,167.301,53.976,160.002
C05216=1015.796,178.403,374.023,167.298,53.987,160.004
C05217=1015.791,178.154,374.043,167.293,53.998,160.005
C05218=1015.787,177.906,374.064,167.289,54.009,160.006
C05219=1015.782,177.656,374.085,167.285,54.019,160.007
C05220=1015.777,177.407,374.106,167.280,54.030,160.009
C05221=1015.772,177.158,374.127,167.277,54.041,160.010
C05222=1015.768,176.909,374.147,167.273,54.051,160.011
C05223=1015.763,176.660,374.168,167.268,54.062,160.012
C05224=1015.759,176.410,374.189,167.264,54.073,160.014
C05225=1015.754,176.162,374.210,167.260,54.084,160.015
C05226=1015.750,175.912,374.230,167.257,54.095,160.017
C05227=1015.745,175.663,374.250,167.252,54.105,160.018
C05228=1015.741,175.414,374.271,167.248,54.116,160.019
C05229=1015.736,175.165,374.293,167.244,54.127,160.020
C05230=1015.731,174.916,374.313,167.241,54.137,160.022
C05231=1015.727,174.667,374.334,167.236,54.148,160.023
C05232=1015.722,174.418,374.354,167.232,54.159,160.024
C05233=1015.718,174.169,374.375,167.229,54.169,160.026
C05234=1015.713,173.919,374.396,167.225,54.180,160.027
C05235=1015.709,173.671,374.417,167.220,54.191,160.028
C05236=1015.704,173.422,374.438,167.216,54.201,160.029
C05237=1015.699,173.172,374.458,167.213,54.212,160.031
C05238=1015.695,172.923,374.478,167.209,54.223,160.032
C05239=1015.691,172.674,374.499,167.204,54.233,160.033
C05240=1015.686,172.425,374.520,167.201,54.244,160.035
C05241=1015.682,172.176,374.541,167.197,54.255,160.036
C05242=1015.677,171.927,374.561,167.192,54.266,160.037
C05243=1015.673,171.677,374.581,167.190,54.276,160.039
C05244=1015.668,171.428,374.603,167.185,54.287,160.040
C05245=1015.662,171.073,374.632,167.180,54.302,160.042
C05246=1015.656,170.717,374.661,167.174,54.318,160.044
C05247=1015.649,170.362,374.691,167.168,54.333,160.046
C05248=1015.643,170.006,374.720,167.163,54.348,160.048
C05249=1015.638,169.757,374.740,167.159,54.358,160.049
C05250=1015.634,169.508,374.761,167.155,54.370,160.050
C05251=1015.629,169.259,374.781,167.152,54.380,160.052
C05252=1015.625,169.010,374.802,167.147,54.391,160.053
C05253=1015.621,168.760,374.823,167.144,54.402,160.054
C05254=1015.616,168.512,374.843,167.140,54.412,160.056
C05255=1015.612,168.263,374.863,167.136,54.423,160.057
C05256=1015.607,168.013,374.883,167.133,54.434,160.058
C05257=1015.603,167.764,374.904,167.128,54.444,160.060
C05258=1015.599,167.515,374.925,167.125,54.454,160.061
C05259=1015.594,167.266,374.945,167.121,54.466,160.062
C05260=1015.590,167.016,374.966,167.117,54.476,160.064
C05261=1015.585,166.768,374.986,167.113,54.487,160.065
C05262=1015.581,166.518,375.006,167.109,54.497,160.066
C05263=1015.577,166.269,375.027,167.106,54.508,160.068
C05264=1015.572,166.021,375.047,167.102,54.519,160.069
C05265=1015.568,165.771,375.068,167.099,54.529,160.070
C05266=1015.563,165.522,375.088,167.095,54.540,160.072
C05267=1015.559,165.272,375.109,167.091,54.551,160.073
C05268=1015.555,165.024,375.129,167.087,54.561,160.074
C05269=1015.551,164.775,375.149,167.084,54.572,160.075
C05270=1015.546,164.525,375.170,167.080,54.583,160.077
C05271=1015.542,164.277,375.190,167.077,54.593,160.078
C05272=1015.538,164.027,375.211,167.072,54.604,160.079
C05273=1015.533,163.778,375.231,167.069,54.614,160.081
C05274=1015.529,163.529,375.251,167.065,54.625,160.082
C05275=1015.525,163.279,375.272,167.062,54.636,160.084
C05276=1015.520,163.031,375.292,167.057,54.646,160.085
C05277=1015.517,162.782,375.312,167.054,54.657,160.086
C05278=1015.511,162.533,375.333,167.050,54.668,160.088
C05279=1015.508,162.283,375.353,167.047,54.678,160.089
C05280=1015.503,162.035,375.373,167.043,54.689,160.090
C05281=1015.499,161.785,375.393,167.039,54.699,160.091
C05282=1015.495,161.536,375.414,167.036,54.711,160.093
C05283=1015.491,161.287,375.434,167.032,54.721,160.094
C05284=1015.486,161.037,375.455,167.028,54.731,160.095
C05285=1015.483,160.826,375.471,167.025,54.741,160.097
C05286=1015.479,160.615,375.488,167.022,54.749,160.098
C05287=1015.476,160.404,375.506,167.019,54.758,160.099
C05288=1015.472,160.192,375.522,167.017,54.767,160.100
C05289=1015.468,159.981,375.540,167.013,54.776,160.101
C05290=1015.465,159.769,375.557,167.010,54.785,160.102
C05291=1015.461,159.558,375.575,167.007,54.795,160.103
C05292=1015.457,159.346,375.591,167.004,54.803,160.104
C05293=1015.454,159.097,375.612,167.000,54.813,160.106
C05294=1015.449,158.847,375.632,166.997,54.825,160.107
C05295=1015.445,158.598,375.652,166.993,54.835,160.109
C05296=1015.441,158.349,375.673,166.990,54.845,160.110
C05297=1015.436,158.100,375.692,166.986,54.856,160.111
C05298=1015.432,157.851,375.712,166.982,54.868,160.113
C05299=1015.427,157.602,375.731,166.979,54.878,160.114
C05300=1015.422,157.352,375.751,166.975,54.889,160.115
C05301=1015.418,157.103,375.771,166.972,54.900,160.117
C05302=1015.414,156.854,375.790,166.968,54.911,160.118
C05303=1015.409,156.605,375.810,166.965,54.921,160.120
C05304=1015.405,156.355,375.831,166.961,54.932,160.121
C05305=1015.401,156.106,375.850,166.958,54.943,160.122
C05306=1015.396,155.857,375.870,166.954,54.954,160.124
C05307=1015.392,155.608,375.889,166.951,54.965,160.125
C05308=1015.387,155.359,375.909,166.947,54.975,160.126
C05309=1015.382,155.078,375.931,166.944,54.988,160.128
C05310=1015.377,154.798,375.953,166.939,54.999,160.129
C05311=1015.372,154.517,375.975,166.936,55.012,160.131
C05312=1015.368,154.237,375.997,166.931,55.024,160.133
C05313=1015.363,153.988,376.016,166.927,55.035,160.134
C05314=1015.358,153.738,376.036,166.924,55.046,160.135
C05315=1015.354,153.489,376.056,166.921,55.056,160.137
C05316=1015.350,153.240,376.075,166.917,55.067,160.138
C05317=1015.346,152.991,376.095,166.914,55.078,160.140
C05318=1015.342,152.742,376.115,166.910,55.089,160.141
C05319=1015.337,152.492,376.134,166.907,55.099,160.142
C05320=1015.332,152.243,376.154,166.903,55.111,160.144
C05321=1015.328,151.994,376.173,166.900,55.121,160.145
C05322=1015.324,151.745,376.193,166.896,55.132,160.146
C05323=1015.319,151.496,376.212,166.893,55.143,160.148
C05324=1015.314,151.247,376.231,166.889,55.154,160.149
C05325=1015.310,150.998,376.251,166.886,55.165,160.151
C05326=1015.305,150.748,376.270,166.882,55.175,160.152
C05327=1015.301,150.499,376.289,166.879,55.186,160.153
C05328=1015.296,150.250,376.309,166.875,55.197,160.155
C05329=1015.292,150.001,376.328,166.873,55.208,160.156
C05330=1015.288,149.751,376.348,166.868,55.219,160.157
C05331=1015.283,149.502,376.367,166.865,55.229,160.159
C05332=1015.279,149.253,376.386,166.863,55.240,160.160
C05333=1015.275,149.004,376.405,166.858,55.251,160.162
C05334=1015.270,148.754,376.425,166.856,55.262,160.163
C05335=1015.266,148.505,376.445,166.852,55.273,160.165
C05336=1015.261,148.256,376.464,166.848,55.283,160.166
C05337=1015.257,148.006,376.483,166.845,55.295,160.167
C05338=1015.253,147.757,376.502,166.842,55.305,160.169
C05339=1015.248,147.508,376.521,166.839,55.316,160.170
C05340=1015.244,147.259,376.541,166.835,55.327,160.172
C05341=1015.240,147.010,376.560,166.832,55.338,160.173
C05342=1015.235,146.761,376.579,166.828,55.349,160.174
C05343=1015.231,146.512,376.598,166.825,55.359,160.176
C05344=1015.227,146.262,376.617,166.822,55.370,160.177
C05345=1015.222,146.013,376.637,166.818,55.381,160.179
C05346=1015.217,145.764,376.656,166.815,55.392,160.180
C05347=1015.213,145.515,376.674,166.811,55.403,160.181
C05348=1015.209,145.266,376.694,166.808,55.414,160.183
C05349=1015.205,145.016,376.713,166.805,55.424,160.184
C05350=1015.200,144.767,376.731,166.802,55.436,160.186
C05351=1015.195,144.517,376.751,166.799,55.446,160.187
C05352=1015.191,144.268,376.770,166.795,55.458,160.189
C05353=1015.186,144.019,376.789,166.792,55.468,160.190
C05354=1015.182,143.769,376.808,166.788,55.479,160.191
C05355=1015.177,143.520,376.827,166.785,55.490,160.193
C05356=1015.173,143.271,376.845,166.781,55.501,160.194
C05357=1015.168,143.022,376.865,166.779,55.512,160.196
C05358=1015.164,142.772,376.884,166.776,55.522,160.197
C05359=1015.159,142.524,376.902,166.772,55.534,160.198
C05360=1015.155,142.274,376.921,166.769,55.544,160.200
C05361=1015.151,142.025,376.941,166.765,55.555,160.201
C05362=1015.146,141.775,376.959,166.762,55.566,160.203
C05363=1015.142,141.527,376.978,166.759,55.577,160.204
C05364=1015.138,141.277,376.997,166.756,55.588,160.206
C05365=1015.133,141.029,377.016,166.753,55.599,160.207
C05366=1015.129,140.779,377.034,166.749,55.609,160.208
C05367=1015.125,140.530,377.054,166.746,55.621,160.210
C05368=1015.120,140.281,377.072,166.743,55.631,160.211
C05369=1015.116,140.031,377.091,166.739,55.642,160.212
C05370=1015.111,139.782,377.110,166.736,55.653,160.214
C05371=1015.107,139.533,377.128,166.733,55.663,160.215
C05372=1015.102,139.284,377.148,166.729,55.674,160.217
C05373=1015.097,139.003,377.168,166.726,55.687,160.218
C05374=1015.092,138.722,377.190,166.723,55.699,160.220
C05375=1015.087,138.442,377.211,166.719,55.711,160.221
C05376=1015.083,138.162,377.232,166.716,55.723,160.223
C05377=1015.079,137.912,377.251,166.713,55.734,160.225
C05378=1015.074,137.663,377.269,166.709,55.745,160.226
C05379=1015.070,137.413,377.288,166.706,55.756,160.228
C05380=1015.065,137.164,377.306,166.703,55.766,160.229
C05381=1015.061,136.915,377.326,166.699,55.778,160.230
C05382=1015.056,136.666,377.344,166.696,55.788,160.232
C05383=1015.052,136.416,377.363,166.694,55.799,160.233
C05384=1015.047,136.167,377.381,166.690,55.810,160.235
C05385=1015.043,135.918,377.400,166.687,55.821,160.236
C05386=1015.039,135.669,377.418,166.685,55.832,160.238
C05387=1015.035,135.419,377.437,166.680,55.843,160.239
C05388=1015.030,135.170,377.455,166.677,55.853,160.240
C05389=1015.025,134.921,377.473,166.674,55.865,160.242
C05390=1015.021,134.671,377.492,166.671,55.875,160.243
C05391=1015.016,134.422,377.511,166.669,55.887,160.245
C05392=1015.012,134.173,377.530,166.665,55.897,160.246
C05393=1015.008,133.924,377.547,166.662,55.908,160.247
C05394=1015.003,133.675,377.566,166.659,55.919,160.249
C05395=1014.999,133.425,377.584,166.655,55.930,160.250
C05396=1014.994,133.176,377.603,166.652,55.941,160.252
C05397=1014.990,132.926,377.621,166.650,55.952,160.253
C05398=1014.985,132.677,377.639,166.647,55.962,160.255
C05399=1014.981,132.429,377.658,166.643,55.974,160.256
C05400=1014.977,132.179,377.677,166.640,55.984,160.258
C05401=1014.972,131.930,377.695,166.637,55.995,160.259
C05402=1014.967,131.680,377.713,166.633,56.006,160.260
C05403=1014.963,131.431,377.732,166.631,56.017,160.262
C05404=1014.959,131.182,377.750,166.628,56.028,160.263
C05405=1014.955,130.932,377.768,166.625,56.038,160.265
C05406=1014.950,130.683,377.786,166.622,56.050,160.266
C05407=1014.945,130.433,377.805,166.619,56.060,160.268
C05408=1014.942,130.185,377.823,166.616,56.071,160.269
C05409=1014.937,129.935,377.841,166.613,56.082,160.271
C05410=1014.933,129.686,377.860,166.609,56.093,160.272
C05411=1014.928,129.436,377.878,166.607,56.103,160.273
C05412=1014.924,129.187,377.896,166.604,56.115,160.275
C05413=1014.919,128.937,377.914,166.600,56.126,160.276
C05414=1014.915,128.688,377.932,166.597,56.136,160.278
C05415=1014.910,128.439,377.950,166.595,56.147,160.279
C05416=1014.905,128.189,377.968,166.591,56.158,160.281
C05417=1014.901,127.940,377.986,166.589,56.170,160.282
C05418=1014.896,127.692,378.004,166.586,56.180,160.284
C05419=1014.892,127.442,378.021,166.582,56.192,160.285
C05420=1014.887,127.192,378.039,166.579,56.202,160.287
C05421=1014.882,126.943,378.058,166.577,56.213,160.288
C05422=1014.878,126.694,378.075,166.573,56.224,160.290
C05423=1014.873,126.445,378.094,166.570,56.235,160.291
C05424=1014.869,126.195,378.111,166.568,56.246,160.293
C05425=1014.865,125.946,378.129,166.564,56.257,160.294
C05426=1014.860,125.697,378.147,166.561,56.268,160.295
C05427=1014.856,125.447,378.165,166.559,56.279,160.297
C05428=1014.851,125.197,378.183,166.555,56.290,160.298
C05429=1014.847,124.949,378.201,166.553,56.301,160.300
C05430=1014.842,124.699,378.219,166.550,56.312,160.301
C05431=1014.838,124.449,378.237,166.547,56.322,160.303
C05432=1014.834,124.201,378.254,166.543,56.334,160.304
C05433=1014.829,123.951,378.272,166.541,56.345,160.306
C05434=1014.825,123.701,378.290,166.538,56.355,160.307
C05435=1014.820,123.453,378.308,166.535,56.366,160.309
C05436=1014.816,123.203,378.326,166.532,56.377,160.310
C05437=1014.810,122.923,378.346,166.529,56.390,160.312
C05438=1014.805,122.643,378.366,166.525,56.402,160.314
C05439=1014.800,122.361,378.385,166.522,56.414,160.315
C05440=1014.796,122.081,378.406,166.518,56.426,160.317
C05441=1014.791,121.832,378.424,166.516,56.437,160.318
C05442=1014.787,121.583,378.442,166.513,56.448,160.320
C05443=1014.782,121.333,378.459,166.510,56.459,160.321
C05444=1014.777,121.084,378.477,166.506,56.470,160.322
C05445=1014.773,120.834,378.494,166.504,56.481,160.324
C05446=1014.769,120.585,378.512,166.501,56.492,160.326
C05447=1014.764,120.336,378.531,166.499,56.502,160.327
C05448=1014.760,120.086,378.548,166.496,56.513,160.328
C05449=1014.755,119.837,378.566,166.492,56.524,160.330
C05450=1014.751,119.588,378.583,166.490,56.535,160.331
C05451=1014.747,119.338,378.601,166.487,56.546,160.333
C05452=1014.742,119.089,378.619,166.484,56.556,160.334
C05453=1014.738,118.840,378.636,166.481,56.567,160.336
C05454=1014.733,118.591,378.654,166.478,56.577,160.337
C05455=1014.729,118.341,378.672,166.476,56.589,160.339
C05456=1014.725,118.092,378.690,166.472,56.600,160.340
C05457=1014.721,117.843,378.707,166.470,56.610,160.342
C05458=1014.716,117.593,378.725,166.467,56.621,160.343
C05459=1014.711,117.344,378.743,166.464,56.632,160.344
C05460=1014.707,117.095,378.760,166.461,56.642,160.346
C05461=1014.702,116.845,378.778,166.458,56.653,160.347
